(* Init ST03_513_B70_2 Führungsschiene  Zuführung Stopper AST (ValveSensor) *)
ST03_513_B70_2.sInit.InstName		:='ST03_513_B70_2';
ST03_513_B70_2.sInit.BitName		:='+8_512_B70.2';
ST03_513_B70_2.sInit.Description	:='Führungsschiene  Zuführung Stopper AST';
ST03_513_B70_2.sInit.SensorType	:=sValveSensorType_WORK;

(* Init ST03_513_B70_3 Führungsschiene  Zuführung Stopper GST (ValveSensor) *)
ST03_513_B70_3.sInit.InstName		:='ST03_513_B70_3';
ST03_513_B70_3.sInit.BitName		:='+8_513_B70.3';
ST03_513_B70_3.sInit.Description	:='Führungsschiene  Zuführung Stopper GST';
ST03_513_B70_3.sInit.SensorType	:=sValveSensorType_INIT;

(* Init ST03_513_B70_4 ISK anwesend am Stoper (DigIn) *)
ST03_513_B70_4.sInit.InstName            :='ST03_513_B70_4';
ST03_513_B70_4.sInit.Description         :='ISK anwesend am Stoper';
ST03_513_B70_4.sInit.BitInName           :='+8-513_B670.4';
ST03_513_B70_4.sInit.HomePosSignal       :=2; (* 0: Signal=Low, 1: Signal=High, 2: always  *)
ST03_513_B70_4.sInit.MaxTime             :=2000;
ST03_513_B70_4.sInit.EnableInEveryMode   :=TRUE;

(* Init ST03_513_B70_5 Übergabeposition Stopper 1 AST (ValveSensor) *)
ST03_513_B70_5.sInit.InstName		:='ST03_513_B70_5';
ST03_513_B70_5.sInit.BitName		:='+8_513_B70.5';
ST03_513_B70_5.sInit.Description	:='Übergabeposition Stopper 1 AST';
ST03_513_B70_5.sInit.SensorType	:=sValveSensorType_WORK;

(* Init ST03_513_B70_6 Übergabeposition Stopper 1 GST (ValveSensor) *)
ST03_513_B70_6.sInit.InstName		:='ST03_513_B70_6';
ST03_513_B70_6.sInit.BitName		:='+8_513_B70.6';
ST03_513_B70_6.sInit.Description	:='Übergabeposition Stopper 1 GST';
ST03_513_B70_6.sInit.SensorType	:=sValveSensorType_INIT;

(* Init ST03_513_B70_7 ISK auf Übergabeposition 1 (DigIn) *)
ST03_513_B70_7.sInit.InstName            :='ST03_513_B70_7';
ST03_513_B70_7.sInit.Description         :='ISK auf Übergabeposition 1';
ST03_513_B70_7.sInit.BitInName           :='+8-513_B670.7';
ST03_513_B70_7.sInit.HomePosSignal       :=2; (* 0: Signal=Low, 1: Signal=High, 2: always  *)
ST03_513_B70_7.sInit.MaxTime             :=2000;
ST03_513_B70_7.sInit.EnableInEveryMode   :=TRUE;


(* Init ST03_514_B71_0 Übergabeposition Stopper 2 AST (ValveSensor) *)
ST03_514_B71_0.sInit.InstName		:='ST03_514_B71_0';
ST03_514_B71_0.sInit.BitName		:='+8_514_B71.0';
ST03_514_B71_0.sInit.Description	:='Übergabeposition Stopper 2 AST';
ST03_514_B71_0.sInit.SensorType	:=sValveSensorType_WORK;

(* Init ST03_514_B71_1 Übergabeposition Stopper 2 GST (ValveSensor) *)
ST03_514_B71_1.sInit.InstName		:='ST03_514_B71_1';
ST03_514_B71_1.sInit.BitName		:='+8_514_B71.1';
ST03_514_B71_1.sInit.Description	:='Übergabeposition Stopper 2 GST';
ST03_514_B71_1.sInit.SensorType	:=sValveSensorType_INIT;

(* Init ST03_514_B71_2 ISK auf Übergabeposition 2 (DigIn) *)
ST03_514_B71_2.sInit.InstName            :='ST03_514_B71_2';
ST03_514_B71_2.sInit.Description         :='ISK auf Übergabeposition 2';
ST03_514_B71_2.sInit.BitInName           :='+8-514_B71.2';
ST03_514_B71_2.sInit.HomePosSignal       :=2; (* 0: Signal=Low, 1: Signal=High, 2: always  *)
ST03_514_B71_2.sInit.MaxTime             :=2000;
ST03_514_B71_2.sInit.EnableInEveryMode   :=TRUE;

(* Init ST03_514_B71_3 Übergabeposition Stopper 3 AST (ValveSensor) *)
ST03_514_B71_3.sInit.InstName		:='ST03_514_B71_3';
ST03_514_B71_3.sInit.BitName		:='+8_514_B71.3';
ST03_514_B71_3.sInit.Description	:='Übergabeposition Stopper 3 AST';
ST03_514_B71_3.sInit.SensorType	:=sValveSensorType_WORK;

(* Init ST03_514_B71_4 Übergabeposition Stopper 3 GST (ValveSensor) *)
ST03_514_B71_4.sInit.InstName		:='ST03_514_B71_4';
ST03_514_B71_4.sInit.BitName		:='+8_514_B71.4';
ST03_514_B71_4.sInit.Description	:='Übergabeposition Stopper 3 GST';
ST03_514_B71_4.sInit.SensorType	:=sValveSensorType_INIT;

(* Init ST03_514_B71_5 ISK auf Übergabeposition 3 (DigIn) *)
ST03_514_B71_5.sInit.InstName            :='ST03_514_B71_5';
ST03_514_B71_5.sInit.Description         :='ISK auf Übergabeposition 3';
ST03_514_B71_5.sInit.BitInName           :='+8-514_B71.5';
ST03_514_B71_5.sInit.HomePosSignal       :=2; (* 0: Signal=Low, 1: Signal=High, 2: always  *)
ST03_514_B71_5.sInit.MaxTime             :=2000;
ST03_514_B71_5.sInit.EnableInEveryMode   :=TRUE;

(* Init ST03_514_B71_6 ISK auf Übergabeposition 4 (DigIn) *)
ST03_514_B71_6.sInit.InstName            :='ST03_514_B71_6';
ST03_514_B71_6.sInit.Description         :='ISK auf Übergabeposition 4';
ST03_514_B71_6.sInit.BitInName           :='+8-514_B71.6';
ST03_514_B71_6.sInit.HomePosSignal       :=2; (* 0: Signal=Low, 1: Signal=High, 2: always  *)
ST03_514_B71_6.sInit.MaxTime             :=2000;
ST03_514_B71_6.sInit.EnableInEveryMode   :=TRUE;

(* Init ST03_514_B71_7 Führungsschiene frei zum schwenken (DigIn) *)
ST03_514_B71_7.sInit.InstName            :='ST03_514_B71_7';
ST03_514_B71_7.sInit.Description         :='Führungsschiene frei zum schwenken';
ST03_514_B71_7.sInit.BitInName           :='+8-514_B71.7';
ST03_514_B71_7.sInit.HomePosSignal       :=2; (* 0: Signal=Low, 1: Signal=High, 2: always  *)
ST03_514_B71_7.sInit.MaxTime             :=2000;
ST03_514_B71_7.sInit.EnableInEveryMode   :=TRUE;

(* Init ST03_515_Y72_0   ISK Klemmer 1 AST/GST (Valve) *)
ST03_515_Y72_0.sInit.InstName            :='ST03_515_Y72_0';
ST03_515_Y72_0.sInit.BitName            :='+8-515_Y72.0';
ST03_515_Y72_0.sInit.Description         :=' ISK Klemmer 1 AST/GST';
ST03_515_Y72_0.sInit.HomePosDefine       :=HOME_ALWAYS;
ST03_515_Y72_0.sInit.InitDescription     :='GS auf';
ST03_515_Y72_0.sInit.WorkDescription     :='AS zu';
(*ST03_515_Y72_0.sInit.InitDescription     :='GS zu';
ST03_515_Y72_0.sInit.WorkDescription     :='AS auf';*)
ST03_515_Y72_0.sInit.DampBothTime        :=200;
ST03_515_Y72_0.sInit.KindOfValve         :='A';
ST03_515_Y72_0.sInit.MaxTime             :=2000;

(* Init ST03_515_Y72_1  Rinne schwenkern  AST/GST (Valve) *)
ST03_515_Y72_1.sInit.InstName            :='ST03_515_Y72_1';
ST03_515_Y72_1.sInit.BitName            :='+8-515_Y72.1';
ST03_515_Y72_1.sInit.Description         :=' Rinne schwenkern AST/GST';
ST03_515_Y72_1.sInit.HomePosDefine       :=HOME_ALWAYS;
ST03_515_Y72_1.sInit.InitDescription     :='GS 0 Grad';
ST03_515_Y72_1.sInit.WorkDescription     :='AS 180 Grad';
ST03_515_Y72_1.sInit.DampBothTime        :=200;
ST03_515_Y72_1.sInit.KindOfValve         :='A';
ST03_515_Y72_1.sInit.MaxTime             :=2000;

(* Init ST03_515_Y72_2  Führungsschiene  Zuführung Vereinzler   AST/GST (Valve) *)
ST03_515_Y72_2.sInit.InstName            :='ST03_515_Y72_2';
ST03_515_Y72_2.sInit.BitName            :='+8-515_Y72.2';
ST03_515_Y72_2.sInit.Description         :=' Führungsschiene  Zuführung Vereinzler AST/GST';
ST03_515_Y72_2.sInit.HomePosDefine       :=HOME_ALWAYS;
ST03_515_Y72_2.sInit.InitDescription     :='GS auf';
ST03_515_Y72_2.sInit.WorkDescription     :='AS zu';
ST03_515_Y72_2.sInit.DampBothTime        :=200;
ST03_515_Y72_2.sInit.KindOfValve         :='A';
ST03_515_Y72_2.sInit.MaxTime             :=2000;

(* Init ST03_515_Y72_3  Führungsschiene  Zuführung Stopper   AST/GST (Valve) *)
ST03_515_Y72_3.sInit.InstName            :='ST03_515_Y72_3';
ST03_515_Y72_3.sInit.BitName            :='+8-515_Y72.3';
ST03_515_Y72_3.sInit.Description         :=' Führungsschiene  Zuführung Stopper AST/GST';
ST03_515_Y72_3.sInit.HomePosDefine       :=HOME_ALWAYS;
ST03_515_Y72_3.sInit.InitDescription     :='GS ausfahren';
ST03_515_Y72_3.sInit.WorkDescription     :='AS einfahren';
ST03_515_Y72_3.sInit.DampBothTime        :=200;
ST03_515_Y72_3.sInit.KindOfValve         :='A';
ST03_515_Y72_3.sInit.MaxTime             :=2000;

(* Init ST03_515_Y72_4  Übergabeposition Stopper 1   AST/GST (Valve) *)
ST03_515_Y72_4.sInit.InstName            :='ST03_515_Y72_4';
ST03_515_Y72_4.sInit.BitName            :='+8-515_Y72.4';
ST03_515_Y72_4.sInit.Description         :=' Übergabeposition Stopper 1 AST/GST';
ST03_515_Y72_4.sInit.HomePosDefine       :=HOME_ALWAYS;
ST03_515_Y72_4.sInit.InitDescription     :='GS ausfahren';
ST03_515_Y72_4.sInit.WorkDescription     :='AS einfahren';
ST03_515_Y72_4.sInit.DampBothTime        :=200;
ST03_515_Y72_4.sInit.KindOfValve         :='A';
ST03_515_Y72_4.sInit.MaxTime             :=2000;

(* Init ST03_515_Y72_5  Übergabeposition Stopper 2   AST/GST (Valve) *)
ST03_515_Y72_5.sInit.InstName            :='ST03_515_Y72_5';
ST03_515_Y72_5.sInit.BitName            :='+8-515_Y72.5';
ST03_515_Y72_5.sInit.Description         :=' Übergabeposition Stopper 2 AST/GST';
ST03_515_Y72_5.sInit.HomePosDefine       :=HOME_ALWAYS;
ST03_515_Y72_5.sInit.InitDescription     :='GS ausfahren';
ST03_515_Y72_5.sInit.WorkDescription     :='AS einfahren';
ST03_515_Y72_5.sInit.DampBothTime        :=200;
ST03_515_Y72_5.sInit.KindOfValve         :='A';
ST03_515_Y72_5.sInit.MaxTime             :=2000;

(* Init ST03_515_Y72_6  Übergabeposition Stopper 3   AST/GST (Valve) *)
ST03_515_Y72_6.sInit.InstName            :='ST03_515_Y72_6';
ST03_515_Y72_6.sInit.BitName            :='+8-515_Y72.6';
ST03_515_Y72_6.sInit.Description         :=' Übergabeposition Stopper 3 AST/GST';
ST03_515_Y72_6.sInit.HomePosDefine       :=HOME_ALWAYS;
ST03_515_Y72_6.sInit.InitDescription     :='GS ausfahren';
ST03_515_Y72_6.sInit.WorkDescription     :='AS einfahren';
ST03_515_Y72_6.sInit.DampBothTime        :=200;
ST03_515_Y72_6.sInit.KindOfValve         :='A';
ST03_515_Y72_6.sInit.MaxTime             :=2000;
END_ACTION
ACTION Init_88pol:
(*Rüstsatz 88 pol==================================================================================*)

(* Init ST03_501_B69_0 Zuführung  frei zum Ablegen ISK SP Maschine (DigIn) *)
ST03_501_B69_0.sInit.InstName            :='ST03_501_B69_0';
ST03_501_B69_0.sInit.Description         :='frei zum Ablegen ISK SP Maschine';
ST03_501_B69_0.sInit.BitInName           :='+8-501_B69.0';
ST03_501_B69_0.sInit.HomePosSignal       :=2; (* 0: Signal=Low, 1: Signal=High, 2: always  *)
ST03_501_B69_0.sInit.MaxTime             :=2000;
ST03_501_B69_0.sInit.EnableInEveryMode   :=TRUE;

(* Init ST03_501_B69_1 Zuführung Vereinzler AST (ValveSensor) *)
ST03_501_B69_1.sInit.InstName		:='ST03_501_B69_1';
ST03_501_B69_1.sInit.BitName		:='+8_501_B69.1';
ST03_501_B69_1.sInit.Description	:='Zuführung Vereinzler AST';
ST03_501_B69_1.sInit.SensorType	:=sValveSensorType_WORK;

(* Init ST03_501_B69_2 Zuführung Vereinzler GST (ValveSensor) *)
ST03_501_B69_2.sInit.InstName		:='ST03_501_B69_2';
ST03_501_B69_2.sInit.BitName		:='+8_501_B69.2';
ST03_501_B69_2.sInit.Description	:='Zuführung Vereinzler GST';
ST03_501_B69_2.sInit.SensorType	:=sValveSensorType_INIT;

(* Init ST03_501_B69_3 Zuführung Stopper AST (ValveSensor) *)
ST03_501_B69_3.sInit.InstName		:='ST03_501_B69_3';
ST03_501_B69_3.sInit.BitName		:='+8_501_B69.3';
ST03_501_B69_3.sInit.Description	:='Zuführung Stopper AST';
ST03_501_B69_3.sInit.SensorType	:=sValveSensorType_WORK;

(* Init ST03_501_B69_4 Zuführung Stopper GST (ValveSensor) *)
ST03_501_B69_4.sInit.InstName		:='ST03_501_B69_4';
ST03_501_B69_4.sInit.BitName		:='+8_501_B69.4';
ST03_501_B69_4.sInit.Description	:='Zuführung Stopper GST';
ST03_501_B69_4.sInit.SensorType	:=sValveSensorType_INIT;

(* Init ST03_501_B69_5 ISK anwesend am Vereinzler (DigIn) *)
ST03_501_B69_5.sInit.InstName            :='ST03_501_B69_5';
ST03_501_B69_5.sInit.Description         :='ISK anwesend am Vereinzler';
ST03_501_B69_5.sInit.BitInName           :='+8-501_B69.5';
ST03_501_B69_5.sInit.HomePosSignal       :=2; (* 0: Signal=Low, 1: Signal=High, 2: always  *)
ST03_501_B69_5.sInit.MaxTime             :=2000;
ST03_501_B69_5.sInit.EnableInEveryMode   :=TRUE;

(* Init ST03_501_B69_6 ISK anwesend am Stopper (DigIn) *)
ST03_501_B69_6.sInit.InstName            :='ST03_501_B69_6';
ST03_501_B69_6.sInit.Description         :='ISK anwesend am Stopper';
ST03_501_B69_6.sInit.BitInName           :='+8-501_B69.6';
ST03_501_B69_6.sInit.HomePosSignal       :=2; (* 0: Signal=Low, 1: Signal=High, 2: always  *)
ST03_501_B69_6.sInit.MaxTime             :=2000;
ST03_501_B69_6.sInit.EnableInEveryMode   :=TRUE;

(* Init ST03_501_B69_7 ISK auf Abholposition Robi (DigIn) *)
ST03_501_B69_7.sInit.InstName            :='ST03_501_B69_7';
ST03_501_B69_7.sInit.Description         :='ISK auf Abholposition Robi';
ST03_501_B69_7.sInit.BitInName           :='+8-501_B69.7';
ST03_501_B69_7.sInit.HomePosSignal       :=2; (* 0: Signal=Low, 1: Signal=High, 2: always  *)
ST03_501_B69_7.sInit.MaxTime             :=2000;
ST03_501_B69_7.sInit.EnableInEveryMode   :=TRUE;

(* Init ST03_502_B70_0 ISK Lageerkennung(DigIn) *)
ST03_502_B70_0.sInit.InstName            :='ST03_502_B70_0';
ST03_502_B70_0.sInit.Description         :='ISK Lageerkennung';
ST03_502_B70_0.sInit.BitInName           :='+8-502_B70.0';
ST03_502_B70_0.sInit.HomePosSignal       :=2; (* 0: Signal=Low, 1: Signal=High, 2: always  *)
ST03_502_B70_0.sInit.MaxTime             :=2000;
ST03_502_B70_0.sInit.EnableInEveryMode   :=TRUE;

(* Init ST03_502_Y70_1  Zuführung  Vereinzler AST/GST (Valve) *)
ST03_502_Y70_1.sInit.InstName            :='ST03_502_Y70_1';
ST03_502_Y70_1.sInit.BitName            :='+8-502_Y70.1';
ST03_502_Y70_1.sInit.Description         :=' Zuführung Vereinzler AST/GST';
ST03_502_Y70_1.sInit.HomePosDefine       :=HOME_ALWAYS;
ST03_502_Y70_1.sInit.InitDescription     :='GS einfahren';
ST03_502_Y70_1.sInit.WorkDescription     :='AS ausfahren';
ST03_502_Y70_1.sInit.DampBothTime        :=200;
ST03_502_Y70_1.sInit.KindOfValve         :='A';
ST03_502_Y70_1.sInit.MaxTime             :=2000;

(* Init ST03_502_Y70_2  Zuführung  Stopper AST/GST (Valve) *)
ST03_502_Y70_2.sInit.InstName            :='ST03_502_Y70_2';
ST03_502_Y70_2.sInit.BitName            :='+8-502_Y70.2';
ST03_502_Y70_2.sInit.Description         :=' Zuführung Stopper AST/GST';
ST03_502_Y70_2.sInit.HomePosDefine       :=HOME_ALWAYS;
ST03_502_Y70_2.sInit.InitDescription     :='GS ausfahren';
ST03_502_Y70_2.sInit.WorkDescription     :='AS einfahren';
ST03_502_Y70_2.sInit.DampBothTime        :=200;
ST03_502_Y70_2.sInit.KindOfValve         :='A';
ST03_502_Y70_2.sInit.MaxTime             :=2000;
END_ACTION
ACTION Init_88polAMG:
(*Rüstsatz 88 pol AMG==================================================================================*)

(* Init ST03_521_B69_0 Zuführung  frei zum Ablegen ISK SP Maschine (DigIn) *)
ST03_521_B69_0.sInit.InstName            :='ST03_521_B69_0';
ST03_521_B69_0.sInit.Description         :='frei zum Ablegen ISK SP Maschine';
ST03_521_B69_0.sInit.BitInName           :='+8-521_B69.0';
ST03_521_B69_0.sInit.HomePosSignal	:=2; (* 0: Signal=Low, 1: Signal=High, 2: always  *)
ST03_521_B69_0.sInit.MaxTime             :=2000;
ST03_521_B69_0.sInit.EnableInEveryMode   :=TRUE;

(* Init ST03_521_B69_1 Zuführung Vereinzler eingefahren GST (ValveSensor) *)
ST03_521_B69_1.sInit.InstName		:='ST03_521_B69_1';
ST03_521_B69_1.sInit.BitName		:='+8_521_B69.1';
ST03_521_B69_1.sInit.Description	:=' Vereinzler eingefahren GST';
ST03_521_B69_1.sInit.SensorType	:=sValveSensorType_INIT;

(* Init ST03_521_B69_2 Zuführung Vereinzler ausgefahren AST (ValveSensor) *)
ST03_521_B69_2.sInit.InstName		:='ST03_521_B69_2';
ST03_521_B69_2.sInit.BitName		:='+8_521_B69.2';
ST03_521_B69_2.sInit.Description	:=' Vereinzler ausgefahren AST';
ST03_521_B69_2.sInit.SensorType	:=sValveSensorType_WORK;

(* Init ST03_521_B69_3 Zuführung Stopper eingefahren AST (ValveSensor) *)
ST03_521_B69_3.sInit.InstName		:='ST03_521_B69_3';
ST03_521_B69_3.sInit.BitName		:='+8_521_B69.3';
ST03_521_B69_3.sInit.Description	:='Stopper eingefahren AST';
ST03_521_B69_3.sInit.SensorType	:=sValveSensorType_WORK;

(* Init ST03_521_B69_4 Zuführung Stopper ausgefahren GST (ValveSensor) *)
ST03_521_B69_4.sInit.InstName		:='ST03_521_B69_4';
ST03_521_B69_4.sInit.BitName		:='+8_521_B69.4';
ST03_521_B69_4.sInit.Description	:='Stopper ausgefahren GST';
ST03_521_B69_4.sInit.SensorType	:=sValveSensorType_INIT;;

(* Init ST03_521_B69_6 ISK anwesend am Stopper (DigIn) *)
ST03_521_B69_6.sInit.InstName            :='ST03_521_B69_6';
ST03_521_B69_6.sInit.Description         :='ISK anwesend am Stopper';
ST03_521_B69_6.sInit.BitInName           :='+8-521_B69.6';
ST03_521_B69_6.sInit.HomePosSignal       :=2; (* 0: Signal=Low, 1: Signal=High, 2: always  *)
ST03_521_B69_6.sInit.MaxTime             :=2000;
ST03_521_B69_6.sInit.EnableInEveryMode   :=TRUE;

(* Init ST03_521_B69_7 ISK Lageerkennung links (DigIn) *)
ST03_521_B69_7.sInit.InstName            :='ST03_521_B69_7';
ST03_521_B69_7.sInit.Description         :='ISK Lageerkennung links';
ST03_521_B69_7.sInit.BitInName           :='+8-521_B69.7';
ST03_521_B69_7.sInit.HomePosSignal       :=2; (* 0: Signal=Low, 1: Signal=High, 2: always  *)
ST03_521_B69_7.sInit.MaxTime             :=2000;
ST03_521_B69_7.sInit.EnableInEveryMode   :=TRUE;

(* Init ST03_522_B70_0 SK Lageerkennung rechts(DigIn) *)
ST03_522_B70_0.sInit.InstName            :='ST03_522_B70_0';
ST03_522_B70_0.sInit.Description         :='ISK Lageerkennung rechts';
ST03_522_B70_0.sInit.BitInName           :='+8-522_B70.0';
ST03_522_B70_0.sInit.HomePosSignal       :=2; (* 0: Signal=Low, 1: Signal=High, 2: always  *)
ST03_522_B70_0.sInit.MaxTime             :=2000;
ST03_522_B70_0.sInit.EnableInEveryMode   :=TRUE;

(* Init ST03_522_Y70_1   Zuführung  Vereinzler AST/GST (Valve) *)
ST03_522_Y70_1.sInit.InstName            :='ST03_522_Y70_1';
ST03_522_Y70_1.sInit.BitName            :='+8-522_Y70.1';
ST03_522_Y70_1.sInit.Description         :=' Zuführung Vereinzler AST/GST';
ST03_522_Y70_1.sInit.HomePosDefine       :=HOME_ALWAYS;
ST03_522_Y70_1.sInit.InitDescription     :='GS einfahren';
ST03_522_Y70_1.sInit.WorkDescription     :='AS ausfahren';
ST03_522_Y70_1.sInit.DampBothTime        :=200;
ST03_522_Y70_1.sInit.KindOfValve         :='A';
ST03_522_Y70_1.sInit.MaxTime             :=2000;

(* Init ST03_522_Y70_2   Zuführung  Stopper AST/GST (Valve) *)
ST03_522_Y70_2.sInit.InstName            :='ST03_522_Y70_2';
ST03_522_Y70_2.sInit.BitName            :='+8-522_Y70.2';
ST03_522_Y70_2.sInit.Description         :=' Zuführung Stopper AST/GST';
ST03_522_Y70_2.sInit.HomePosDefine       :=HOME_ALWAYS;
ST03_522_Y70_2.sInit.InitDescription     :='GS ausfahren';
ST03_522_Y70_2.sInit.WorkDescription     :='AS einfahren';
ST03_522_Y70_2.sInit.DampBothTime        :=200;
ST03_522_Y70_2.sInit.KindOfValve         :='A';
ST03_522_Y70_2.sInit.MaxTime             :=2000;
END_ACTION
ACTION Init_92pol:
(*Rüstsatz 92pol*)
(* Init ST03_444_B69_0 Förderbandeinheit  Zuführung Vereinzler AST (ValveSensor) *)
ST03_444_B69_0.sInit.InstName            :='ST03_444_B69_0';
ST03_444_B69_0.sInit.BitName            :='+8_444_B69.0';
ST03_444_B69_0.sInit.Description         :='Förderbandeinheit  Zuführung Vereinzler AST';
ST03_444_B69_0.sInit.SensorType          :=sValveSensorType_INIT;

(* Init ST03_444_B69_1 Förderbandeinheit  Zuführung Vereinzler GST (ValveSensor) *)
ST03_444_B69_1.sInit.InstName            :='ST03_444_B69_1';
ST03_444_B69_1.sInit.BitName            :='+8_444_B69.1';
ST03_444_B69_1.sInit.Description         :='Förderbandeinheit  Zuführung Vereinzler GST';
ST03_444_B69_1.sInit.SensorType          :=sValveSensorType_WORK;

(* Init ST03_444_B69_2 Förderbandeinheit  Zuführung Stopper AST (ValveSensor) *)
ST03_444_B69_2.sInit.InstName            :='ST03_444_B69_2';
ST03_444_B69_2.sInit.BitName            :='+8_444_B69.2';
ST03_444_B69_2.sInit.Description         :='Förderband linke Zuführung Stopper AST';
ST03_444_B69_2.sInit.SensorType          :=sValveSensorType_INIT;

(* Init ST03_444_B69_3 Förderbandeinheit  Zuführung Stopper GST (ValveSensor) *)
ST03_444_B69_3.sInit.InstName            :='ST03_444_B69_3';
ST03_444_B69_3.sInit.BitName            :='+8_444_B69.3';
ST03_444_B69_3.sInit.Description         :='Förderband linke Zuführung Stopper GST';
ST03_444_B69_3.sInit.SensorType          :=sValveSensorType_WORK;

(* Init ST03_444_B69_4  Zuführung  frei zum Ablegen ISK SP Maschine Pos.1 (DigIn) *)
ST03_444_B69_4.sInit.InstName            :='ST03_444_B69_4';
ST03_444_B69_4.sInit.Description         :='Zuführung links frei zum Ablegen ISK SP Maschine Pos1';
ST03_444_B69_4.sInit.BitInName           :='+8-444_B69.4';
ST03_444_B69_4.sInit.HomePosSignal       :=2; (* 0: Signal=Low, 1: Signal=High, 2: always  *)
ST03_444_B69_4.sInit.MaxTime             :=2000;
ST03_444_B69_4.sInit.EnableInEveryMode   :=TRUE;

(* Init ST03_444_B69_7  ISK anwesend am Vereinzler (DigIn) *)
ST03_444_B69_7.sInit.InstName            :='ST03_444_B69_7';
ST03_444_B69_7.sInit.Description         :='ISK anwesend am Vereinzler';
ST03_444_B69_7.sInit.BitInName           :='+8-444_B69.7';
ST03_444_B69_7.sInit.HomePosSignal       :=2; (* 0: Signal=Low, 1: Signal=High, 2: always  *)
ST03_444_B69_7.sInit.MaxTime             :=2000;
ST03_444_B69_7.sInit.EnableInEveryMode   :=TRUE;

(* Init ST03_445_B70_1  Züführung  ISK Lageerkennung 1 (DigIn) *)
ST03_445_B70_1.sInit.InstName            :='ST03_445_B70_1';
ST03_445_B70_1.sInit.Description         :='Züführung  ISK Lageerkennung 1';
ST03_445_B70_1.sInit.BitInName           :='+8-445_B70.1';
ST03_445_B70_1.sInit.HomePosSignal       :=2; (* 0: Signal=Low, 1: Signal=High, 2: always  *)
ST03_445_B70_1.sInit.MaxTime             :=2000;
ST03_445_B70_1.sInit.EnableInEveryMode   :=TRUE;

(* Init ST03_445_B70_2  Züführung  ISK Lageerkennung 2 (DigIn) *)
ST03_445_B70_2.sInit.InstName            :='ST03_445_B70_2';
ST03_445_B70_2.sInit.Description         :='Züführung  ISK Lageerkennung 2';
ST03_445_B70_2.sInit.BitInName           :='+8-445_B70.2';
ST03_445_B70_2.sInit.HomePosSignal       :=2; (* 0: Signal=Low, 1: Signal=High, 2: always  *)
ST03_445_B70_2.sInit.MaxTime             :=2000;
ST03_445_B70_2.sInit.EnableInEveryMode   :=TRUE;

(* Init ST03_446_B70_4  ISK anwesend Übergabeposition Roboter (DigIn) *)
ST03_446_B70_4.sInit.InstName            :='ST03_446_B70_4';
ST03_446_B70_4.sInit.Description         :='Zuführung ISK auf Übergabeposition Robo Palettierer ';
ST03_446_B70_4.sInit.BitInName           :='+8-446_B70.4';
ST03_446_B70_4.sInit.HomePosSignal       :=2; (* 0: Signal=Low, 1: Signal=High, 2: always  *)
ST03_446_B70_4.sInit.MaxTime             :=2000;
ST03_446_B70_4.sInit.EnableInEveryMode   :=TRUE;

(* Init ST03_446_Y70_5 Förderband  Zuführung Vereinzler (Valve) *)
ST03_446_Y70_5.sInit.InstName            :='ST03_446_Y70_5';
ST03_446_Y70_5.sInit.BitName            :='+8-446_Y70.5';
ST03_446_Y70_5.sInit.Description         :='Förderband  Zuführung Vereinzler';
ST03_446_Y70_5.sInit.HomePosDefine       :=HOME_ALWAYS;
ST03_446_Y70_5.sInit.InitDescription     :='GS einfahren';
ST03_446_Y70_5.sInit.WorkDescription     :='AS ausfahren';
ST03_446_Y70_5.sInit.DampBothTime        :=200;
ST03_446_Y70_5.sInit.KindOfValve         :='A';
ST03_446_Y70_5.sInit.MaxTime             :=2000;

(* Init ST03_446_Y70_6 Förderband  Zuführung Stopper (Valve) *)
ST03_446_Y70_6.sInit.InstName            :='ST03_446_Y70_6';
ST03_446_Y70_6.sInit.BitName            :='+8-446_Y70.6';
ST03_446_Y70_6.sInit.Description         :='Förderband  Zuführung Stopper';
ST03_446_Y70_6.sInit.HomePosDefine       :=HOME_ALWAYS;
ST03_446_Y70_6.sInit.InitDescription     :='GS ausfahren';
ST03_446_Y70_6.sInit.WorkDescription     :='AS einfahren';
ST03_446_Y70_6.sInit.DampBothTime        :=200;
ST03_446_Y70_6.sInit.KindOfValve         :='A';
ST03_446_Y70_6.sInit.MaxTime             :=2000;
END_ACTION
ACTION Init_NOX4pol:
(*Rüstsatz NOX 4 pol==================================================================================*)

(* Init ST03_491_B69_0 Zuführung  frei zum Ablegen ISK SP Maschine (DigIn) *)
ST03_491_B69_0.sInit.InstName            :='ST03_491_B69_0';
ST03_491_B69_0.sInit.Description         :='frei zum Ablegen ISK SP Maschine';
ST03_491_B69_0.sInit.BitInName           :='+8-491_B69.0';
ST03_491_B69_0.sInit.HomePosSignal       :=2; (* 0: Signal=Low, 1: Signal=High, 2: always  *)
ST03_491_B69_0.sInit.MaxTime             :=2000;
ST03_491_B69_0.sInit.EnableInEveryMode   :=TRUE;

(* Init ST03_491_B69_5 ISK anwesend am Stoper (DigIn) *)
ST03_491_B69_5.sInit.InstName            :='ST03_491_B69_5';
ST03_491_B69_5.sInit.Description         :='ISK anwesend am Stoper';
ST03_491_B69_5.sInit.BitInName           :='+8-491_B69.5';
ST03_491_B69_5.sInit.HomePosSignal       :=2; (* 0: Signal=Low, 1: Signal=High, 2: always  *)
ST03_491_B69_5.sInit.MaxTime             :=2000;
ST03_491_B69_5.sInit.EnableInEveryMode   :=TRUE;

(* Init ST03_491_B69_7 SK auf Abholposition Robi (DigIn) *)
ST03_491_B69_7.sInit.InstName            :='ST03_491_B69_7';
ST03_491_B69_7.sInit.Description         :='SK auf Abholposition Robi';
ST03_491_B69_7.sInit.BitInName           :='+8-491_B69.5';
ST03_491_B69_7.sInit.HomePosSignal       :=2; (* 0: Signal=Low, 1: Signal=High, 2: always  *)
ST03_491_B69_7.sInit.MaxTime             :=2000;
ST03_491_B69_7.sInit.EnableInEveryMode   :=TRUE;

(* Init ST03_492_Y70_0  Zuführung Vereinzler AST/GST (Valve) *)
ST03_492_Y70_0.sInit.InstName            :='ST03_492_Y70_0';
ST03_492_Y70_0.sInit.BitName            :='+8-492_Y70.0';
ST03_492_Y70_0.sInit.Description         :='Zuführung Vereinzler AST/GST';
ST03_492_Y70_0.sInit.HomePosDefine       :=HOME_ALWAYS;
ST03_492_Y70_0.sInit.InitDescription     :='GS einfahren';
ST03_492_Y70_0.sInit.WorkDescription     :='AS ausfahren';
ST03_492_Y70_0.sInit.DampBothTime        :=200;
ST03_492_Y70_0.sInit.KindOfValve         :='A';
ST03_492_Y70_0.sInit.MaxTime             :=2000;

(* Init ST03_491_B69_1 Zuführung Vereinzler AST (ValveSensor) *)
ST03_491_B69_1.sInit.InstName		:='ST03_491_B69_1';
ST03_491_B69_1.sInit.BitName		:='+8_491_B69.1';
ST03_491_B69_1.sInit.Description	:='Zuführung  Vereinzler AST';
ST03_491_B69_1.sInit.SensorType	:=sValveSensorType_WORK;

(* Init ST03_491_B69_2 Zuführung Vereinzler GST (ValveSensor) *)
ST03_491_B69_2.sInit.InstName		:='ST03_491_B69_2';
ST03_491_B69_2.sInit.BitName		:='+8_491_B69.2';
ST03_491_B69_2.sInit.Description	:='Zuführung Vereinzler GST';
ST03_491_B69_2.sInit.SensorType	:=sValveSensorType_INIT;

(* Init ST03_492_Y70_1   Zuführung  Stopper AST/GST (Valve) *)
ST03_492_Y70_1.sInit.InstName            :='ST03_492_Y70_1';
ST03_492_Y70_1.sInit.BitName            :='+8-492_Y70.1';
ST03_492_Y70_1.sInit.Description         :=' Zuführung Stopper AST/GST';
ST03_492_Y70_1.sInit.HomePosDefine       :=HOME_ALWAYS;
ST03_492_Y70_1.sInit.InitDescription     :='GS ausfahren';
ST03_492_Y70_1.sInit.WorkDescription     :='AS einfahren';
ST03_492_Y70_1.sInit.DampBothTime        :=200;
ST03_492_Y70_1.sInit.KindOfValve         :='A';
ST03_492_Y70_1.sInit.MaxTime             :=2000;

(* Init ST03_491_B69_3 Zuführung Stopper AST (ValveSensor) *)
ST03_491_B69_3.sInit.InstName		:='ST03_491_B69_3';
ST03_491_B69_3.sInit.BitName		:='+8_491_B69.3';
ST03_491_B69_3.sInit.Description	:='Zuführung Stopper AST';
ST03_491_B69_3.sInit.SensorType	:=sValveSensorType_WORK;

(* Init ST03_491_B69_4 Zuführung Stopper GST (ValveSensor) *)
ST03_491_B69_4.sInit.InstName		:='ST03_491_B69_4';
ST03_491_B69_4.sInit.BitName		:='+8_491_B69.4';
ST03_491_B69_4.sInit.Description	:='Zuführung Stopper GST';
ST03_491_B69_4.sInit.SensorType	:=sValveSensorType_INIT;
END_ACTION
ACTION Init_NOX5_6pol:
(*===============================Rüstsatz NOX 5+6 pol==========================*)

(* Init ST03_4x2_B69_0 Zuführung frei zum Ablegen ISK SP Maschine (DigIn) *)
ST03_4x2_B69_0.sInit.InstName            :='ST03_4x2_B69_0';
ST03_4x2_B69_0.sInit.Description         :='Zuführung frei zum Ablegen ISK SP Maschine';
ST03_4x2_B69_0.sInit.BitInName           :='+8-4x2_B69.0';
ST03_4x2_B69_0.sInit.HomePosSignal       :=2; (* 0: Signal=Low, 1: Signal=High, 2: always  *)
ST03_4x2_B69_0.sInit.MaxTime             :=2000;
ST03_4x2_B69_0.sInit.EnableInEveryMode   :=TRUE;

(* Init ST03_4x2_B69_1 Zuführung Vereinzler GST eingefahren (ValveSensor) *)
ST03_4x2_B69_1.sInit.InstName		:='ST03_4x2_B69_1';
ST03_4x2_B69_1.sInit.BitName		:='+8_4x2_B69.1';
ST03_4x2_B69_1.sInit.Description	:='Zuführung Vereinzler GST';
ST03_4x2_B69_1.sInit.SensorType		:=sValveSensorType_INIT;

(* Init ST03_4x2_B69_2 Zuführung Vereinzler AST ausgefahren (ValveSensor) *)
ST03_4x2_B69_2.sInit.InstName		:='ST03_4x2_B69_2';
ST03_4x2_B69_2.sInit.BitName		:='+8_4x2_B69.2';
ST03_4x2_B69_2.sInit.Description	:='Zuführung Vereinzler AST';
ST03_4x2_B69_2.sInit.SensorType		:=sValveSensorType_WORK;

(* Init ST03_4x2_B69_3 Zuführung Stopper GST eingefahren (ValveSensor) *)
ST03_4x2_B69_3.sInit.InstName		:='ST03_4x2_B69_3';
ST03_4x2_B69_3.sInit.BitName		:='+8_4x2_B69.3';
ST03_4x2_B69_3.sInit.Description	:='Zuführung Stopper AST';
ST03_4x2_B69_3.sInit.SensorType		:=sValveSensorType_WORK;

(* Init ST03_4x2_B69_4 Zuführung Stopper AST ausgefahren (ValveSensor) *)
ST03_4x2_B69_4.sInit.InstName		:='ST03_4x2_B69_4';
ST03_4x2_B69_4.sInit.BitName		:='+8_4x2_B69.4';
ST03_4x2_B69_4.sInit.Description	:='Zuführung Stopper GST';
ST03_4x2_B69_4.sInit.SensorType		:=sValveSensorType_INIT;

(* Init ST03_4x2_B69_5 ISK anwesend am Stopper (DigIn) *)
ST03_4x2_B69_5.sInit.InstName            :='ST03_4x2_B69_5';
ST03_4x2_B69_5.sInit.Description         :='ISK anwesend am Stopper';
ST03_4x2_B69_5.sInit.BitInName           :='+8-4x2_B69.5';
ST03_4x2_B69_5.sInit.HomePosSignal       :=2; (* 0: Signal=Low, 1: Signal=High, 2: always  *)
ST03_4x2_B69_5.sInit.MaxTime             :=2000;
ST03_4x2_B69_5.sInit.EnableInEveryMode   :=TRUE;

(* Init ST03_4x2_B69_6 Zuführung Stopper GST eingefahren (ValveSensor) *)
ST03_4x2_B69_6.sInit.InstName		:='ST03_4x2_B69_6';
ST03_4x2_B69_6.sInit.BitName		:='+8_4x2_B69.6';
ST03_4x2_B69_6.sInit.Description	:='Zuführung Stopper Übergabeposition AST';
ST03_4x2_B69_6.sInit.SensorType		:=sValveSensorType_WORK;

(* Init ST03_4x2_B69_7 Zuführung Stopper AST ausgefahren (ValveSensor) *)
ST03_4x2_B69_7.sInit.InstName		:='ST03_4x2_B69_7';
ST03_4x2_B69_7.sInit.BitName		:='+8_4x2_B69.7';
ST03_4x2_B69_7.sInit.Description	:='Zuführung Stopper Übergabeposition GST';
ST03_4x2_B69_7.sInit.SensorType		:=sValveSensorType_INIT;

(* Init ST03_4x3_B70_0 ISK anwesend Übergabeposition Stopper (DigIn) *)
ST03_4x3_B70_0.sInit.InstName            :='ST03_4x3_B70_0';
ST03_4x3_B70_0.sInit.Description         :='ISK anwesend Übergabeposition Stopper';
ST03_4x3_B70_0.sInit.BitInName           :='+8-4x3_B70.0';
ST03_4x3_B70_0.sInit.HomePosSignal       :=2; (* 0: Signal=Low, 1: Signal=High, 2: always  *)
ST03_4x3_B70_0.sInit.MaxTime             :=2000;
ST03_4x3_B70_0.sInit.EnableInEveryMode   :=TRUE;

(* Init ST03_4x3_B70_1 ISK anwesend Übergabeposition (DigIn) *)
ST03_4x3_B70_1.sInit.InstName            :='ST03_4x3_B70_1';
ST03_4x3_B70_1.sInit.Description         :='ISK anwesend Übergabeposition';
ST03_4x3_B70_1.sInit.BitInName           :='+8-4x3_B70.1';
ST03_4x3_B70_1.sInit.HomePosSignal       :=2; (* 0: Signal=Low, 1: Signal=High, 2: always  *)
ST03_4x3_B70_1.sInit.MaxTime             :=2000;
ST03_4x3_B70_1.sInit.EnableInEveryMode   :=TRUE;

(* Init ST03_4x3_Y70_5  Zuführung Vereinzler AST/GST (Valve) *)
ST03_4x3_Y70_5.sInit.InstName            :='ST03_4x3_Y70_5';
ST03_4x3_Y70_5.sInit.BitName            :='+8-4x3_Y70.5';
ST03_4x3_Y70_5.sInit.Description         :='Zuführung Vereinzler AST/GST';
ST03_4x3_Y70_5.sInit.HomePosDefine       :=HOME_ALWAYS;
ST03_4x3_Y70_5.sInit.InitDescription     :='GS einfahren';
ST03_4x3_Y70_5.sInit.WorkDescription     :='AS ausfahren';
ST03_4x3_Y70_5.sInit.DampBothTime        :=200;
ST03_4x3_Y70_5.sInit.KindOfValve         :='A';
ST03_4x3_Y70_5.sInit.MaxTime             :=2000;

(* Init ST03_4x3_Y70_6   Zuführung Stopper AST/GST (Valve) *)
ST03_4x3_Y70_6.sInit.InstName            :='ST03_4x3_Y70_6';
ST03_4x3_Y70_6.sInit.BitName            :='+8-4x3_Y70.6';
ST03_4x3_Y70_6.sInit.Description         :=' Zuführung Stopper AST/GST';
ST03_4x3_Y70_6.sInit.HomePosDefine       :=HOME_ALWAYS;
ST03_4x3_Y70_6.sInit.InitDescription     :='GS ausfahren';
ST03_4x3_Y70_6.sInit.WorkDescription     :='AS einfahren';
ST03_4x3_Y70_6.sInit.DampBothTime        :=200;
ST03_4x3_Y70_6.sInit.KindOfValve         :='A';
ST03_4x3_Y70_6.sInit.MaxTime             :=2000;

(* Init ST03_4x3_Y70_7   Zuführung Stopper Übergabeposition AST/GST (Valve) *)
ST03_4x3_Y70_7.sInit.InstName            :='ST03_4x3_Y70_7';
ST03_4x3_Y70_7.sInit.BitName            :='+8-4x3_Y70.7';
ST03_4x3_Y70_7.sInit.Description         :=' Zuführung Stopper Übergabeposition AST/GST';
ST03_4x3_Y70_7.sInit.HomePosDefine       :=HOME_ALWAYS;
ST03_4x3_Y70_7.sInit.InitDescription     :='GS ausfahren';
ST03_4x3_Y70_7.sInit.WorkDescription     :='AS einfahren';
ST03_4x3_Y70_7.sInit.DampBothTime        :=200;
ST03_4x3_Y70_7.sInit.KindOfValve         :='A';
ST03_4x3_Y70_7.sInit.MaxTime             :=2000;
END_ACTION

(* POU Stations/ST_08_Palettierer/ST_08__InitFBs/ST08_Init, ST *)
PROGRAM ST08_Init


VAR


END_VAR
(* ----------------------------------------------------------------------------------------- *)
(*Init ST08_180_M1 Abstapeln*)
ST08_180_M1.sConfig.Description			:='Abstapeln';
ST08_180_M1.sConfig.InstName			:='ST08_180_M1';
ST08_180_M1.sConfig.Skalierfaktor		:=360.0 / (EXPT(2,20))	; (*360°/ 20 bit Encoder =0.00034332275390625*)
ST08_180_M1.sConfig.Getriebefaktor		:=10;
ST08_180_M1.sConfig.Modulo				:=FALSE;
ST08_180_M1.sConfig.Pos_Faktor			:=5;				(*Weg bei einer Umdrehung in mm (nach Getriebe)*)
ST08_180_M1.sConfig.maxRpm				:=3500;
ST08_180_M1.sConfig.ModeOfOperation		:=CSP;			(*CSP,CSV,CST,CSTCA muss an der KLemme (Coe-Online 7010.03) eingestellt werden*)
(*(CSP) position mode*)
ST08_180_M1.sConfig.Torque_Limit		:=0;			(*bei 0 ausgeschaltet*)
ST08_180_M1.sConfig.SW_Limit_on			:=TRUE;
ST08_180_M1.sConfig.SW_Limit_min		:=-8;
ST08_180_M1.sConfig.SW_Limit_max		:=185;
ST08_180_M1.sConfig.lr_kp 				:= 800;
ST08_180_M1.sConfig.lr_ki 				:= 100.0;
ST08_180_M1.sConfig.lr_kd 				:= 50;
(* ----------------------------------------------------------------------------------------- *)
(*Init ST08_185_M1 Aufstapeln*)
ST08_185_M1.sConfig.Description		:='Aufstapeln';
ST08_185_M1.sConfig.InstName			:='ST08_185_M1';
ST08_185_M1.sConfig.Skalierfaktor		:=360.0 / (EXPT(2,20))	; (*360°/ 20 bit Encoder =0.00034332275390625*)
ST08_185_M1.sConfig.Getriebefaktor		:=10;
ST08_185_M1.sConfig.Modulo			:=FALSE;
ST08_185_M1.sConfig.Pos_Faktor		:=5;			(*Weg bei einer Umdrehung in mm (nach Getriebe)*)
ST08_185_M1.sConfig.maxRpm			:=3500;
ST08_185_M1.sConfig.ModeOfOperation	:=CSP;		(*CSP,CSV,CST,CSTCA muss an der KLemme (Coe-Online 7010.03) eingestellt werden*)
(*(CSP) position mode*)
ST08_185_M1.sConfig.Torque_Limit		:=0;			(*bei 0 ausgeschaltet*)
ST08_185_M1.sConfig.SW_Limit_on		:=TRUE;
ST08_185_M1.sConfig.SW_Limit_min		:=-8;
ST08_185_M1.sConfig.SW_Limit_max	:=185;
ST08_185_M1.sConfig.lr_kp 				:= 800;
ST08_185_M1.sConfig.lr_ki 				:= 100.0;
ST08_185_M1.sConfig.lr_kd 				:= 50;
(* ----------------------------------------------------------------------------------------- *)
(*Init ST08_190_M1 Tray ausheben*)
ST08_190_M1.sConfig.Description		:='Tray ausheben';
ST08_190_M1.sConfig.InstName			:='ST08_190_M1';
ST08_190_M1.sConfig.Skalierfaktor		:=360.0 / (EXPT(2,20))	; (*360°/ 20 bit Encoder =0.00034332275390625*)
ST08_190_M1.sConfig.Getriebefaktor		:=1;
ST08_190_M1.sConfig.Modulo			:=FALSE;
ST08_190_M1.sConfig.Pos_Faktor		:=5;			(*Weg bei einer Umdrehung in mm (nach Getriebe)*)
ST08_190_M1.sConfig.maxRpm			:=3500;
ST08_190_M1.sConfig.ModeOfOperation	:=CSP;		(*CSP,CSV,CST,CSTCA muss an der KLemme (Coe-Online 7010.03) eingestellt werden*)
(*(CSP) position mode*)
ST08_190_M1.sConfig.Torque_Limit		:=0;			(*bei 0 ausgeschaltet*)
ST08_190_M1.sConfig.SW_Limit_on		:=TRUE;
ST08_190_M1.sConfig.SW_Limit_min		:=-20;
ST08_190_M1.sConfig.SW_Limit_max	:=185;
ST08_190_M1.sConfig.lr_kp 				:= 800;
ST08_190_M1.sConfig.lr_ki 				:= 100.0;
ST08_190_M1.sConfig.lr_kd 				:= 50;
(* ----------------------------------------------------------------------------------------- *)

(* Init ST08_400_B50_0 Traystapel vor Vereinzeler Einlaufband hinten (DigIn) *)
ST08_400_B50_0.sInit.InstName            :='ST08_400_B50_0';
ST08_400_B50_0.sInit.Description         :='Traystapel hinten vor Vereinzeler Einlaufband hinten';
ST08_400_B50_0.sInit.BitInName           :='+8-400_B50.0';
ST08_400_B50_0.sInit.HomePosSignal       :=2; (* 0: Signal=Low, 1: Signal=High, 2: always  *)
ST08_400_B50_0.sInit.MaxTime             :=2000;

(* Init ST08_400_B50_4 Stopper Traystapel Einlaufband hinten rechts GST (ValveSensor) *)
ST08_400_B50_4.sInit.InstName            :='ST08_400_B50_4';
ST08_400_B50_4.sInit.BitName            :='+8_400_B50.4';
ST08_400_B50_4.sInit.Description         :='Stopper Traystapel Einlaufband hinten rechts GST';
ST08_400_B50_4.sInit.SensorType          :=sValveSensorType_INIT;

(* Init ST08_401_B50_5 Traystapel vor Vereinzeler Einlaufband mitte (DigIn) *)
ST08_401_B50_5.sInit.InstName            :='ST08_401_B50_5';
ST08_401_B50_5.sInit.Description         :='Traystapel mitte vor Vereinzeler Einlaufband ';
ST08_401_B50_5.sInit.BitInName           :='+8-401_B50.5';
ST08_401_B50_5.sInit.HomePosSignal       :=2; (* 0: Signal=Low, 1: Signal=High, 2: always  *)
ST08_401_B50_5.sInit.MaxTime             :=2000;

(* Init ST08_401_B51_1 Stopper Traystapel Einlaufband mitte rechts GST (ValveSensor) *)
ST08_401_B51_1.sInit.InstName            :='ST08_401_B51_1';
ST08_401_B51_1.sInit.BitName            :='+8_401_B51.1';
ST08_401_B51_1.sInit.Description         :='Stopper Traystapel Einlaufband mitte rechts GST';
ST08_401_B51_1.sInit.SensorType          :=sValveSensorType_INIT;


(* Init ST08_402_B51_2 Traystapel vor Vereinzeler Einlaufband vorne (DigIn) *)
ST08_402_B51_2.sInit.InstName            :='ST08_402_B51_2';
ST08_402_B51_2.sInit.Description         :='Traystapel vorne vor Vereinzeler Einlaufband ';
ST08_402_B51_2.sInit.BitInName           :='+8-402_B51.2';
ST08_402_B51_2.sInit.HomePosSignal       :=2; (* 0: Signal=Low, 1: Signal=High, 2: always  *)
ST08_402_B51_2.sInit.MaxTime             :=2000;

(*ST08_402_B51_3 Traystapel schieben mitte ausgefahren (ValveSensor)*)
ST08_402_B51_3.sInit.InstName            :='ST08_402_B51_3';
ST08_402_B51_3.sInit.BitName            :='+8_402_B51.3';
ST08_402_B51_3.sInit.Description         :='Traystapel schieben mitte';
ST08_402_B51_3.sInit.SensorType          :=sValveSensorType_INIT;

(* Init ST08_402_B51_4 (* Luftzone 1 *) (DigIn) *)
ST08_402_B51_4.sInit.InstName            :='ST08_402_B51_4';
ST08_402_B51_4.sInit.Description         :='Druckschalter St08 Zone2';
ST08_402_B51_4.sInit.BitInName           :='+8-402_B51.4';
ST08_402_B51_4.sInit.HomePosSignal       :=2; (* 0: Signal=Low, 1: Signal=High, 2: always  *)
ST08_402_B51_4.sInit.MaxTime             :=2000;
ST08_402_B51_4.sInit.EnableInEveryMode   :=TRUE;

(* Init ST08_402_B51_5 (* Luftzone 1 *) (DigIn) *)
ST08_402_B51_5.sInit.InstName            :='ST08_402_B51_5';
ST08_402_B51_5.sInit.Description         :='Druckschalter St08 Zone3';
ST08_402_B51_5.sInit.BitInName           :='+8-402_B51.5';
ST08_402_B51_5.sInit.HomePosSignal       :=2; (* 0: Signal=Low, 1: Signal=High, 2: always  *)
ST08_402_B51_5.sInit.MaxTime             :=2000;
ST08_402_B51_5.sInit.EnableInEveryMode   :=TRUE;

(* Init ST08_402_B51_6 Stopper Traystapel Einlaufband vorne rechts GST (ValveSensor) *)
ST08_402_B51_6.sInit.InstName            :='ST08_402_B51_6';
ST08_402_B51_6.sInit.BitName            :='+8_402_B51.6';
ST08_402_B51_6.sInit.Description         :='Stopper Traystapel Einlaufband vorne rechts GST';
ST08_402_B51_6.sInit.SensorType          :=sValveSensorType_INIT;

(*ST08_402_B51_7 Traystapel schieben vorne ausgefahren (ValveSensor)*)
ST08_402_B51_7.sInit.InstName            :='ST08_402_B51_7';
ST08_402_B51_7.sInit.BitName            :='+8_402_B51.7';
ST08_402_B51_7.sInit.Description         :='Traystapel schieben vorne';
ST08_402_B51_7.sInit.SensorType          :=sValveSensorType_INIT;

(* Init ST08_403_B52_0 Hubstüre 1 AST (ValveSensor) *)
ST08_403_B52_0.sInit.InstName            :='ST08_403_B52_0';
ST08_403_B52_0.sInit.BitName            :='+8_403_B52_0';
ST08_403_B52_0.sInit.Description         :='Hubtüre 1 Einlauf STN8 AST';
ST08_403_B52_0.sInit.SensorType          :=sValveSensorType_WORK;

(* Init ST08_403_B52_1 Hubstüre 1 GST  (ValveSensor) *)
ST08_403_B52_1.sInit.InstName            :='ST08_403_B52_1';
ST08_403_B52_1.sInit.BitName            :='+8_403_B52_1';
ST08_403_B52_1.sInit.Description         :='Hubtüre 1 Einlauf STN8 AST';
ST08_403_B52_1.sInit.SensorType          :=sValveSensorType_INIT;

(* Init ST08_404_B52_2 Traystapel in Ablageposition Isokörper (DigIn) *)
ST08_404_B52_2.sInit.InstName            :='ST08_404_B52_2';
ST08_404_B52_2.sInit.Description         :='Traystapel in Ablageposition Isokörper';
ST08_404_B52_2.sInit.BitInName           :='+8-404_B52.2'; 
ST08_404_B52_2.sInit.HomePosSignal       :=2; (* 0: Signal=Low, 1: Signal=High, 2: always  *)
ST08_404_B52_2.sInit.MaxTime             :=2000;

(* Init ST08_404_B52_3 Traystapel richtig eingelegt Isokörper (DigIn) *)
ST08_404_B52_3.sInit.InstName            :='ST08_404_B52_3';
ST08_404_B52_3.sInit.Description         :='Traystapel richtig eingelegt Isokörper';
ST08_404_B52_3.sInit.BitInName           :='+8-404_B52.3';
ST08_404_B52_3.sInit.HomePosSignal       :=2; (* 0: Signal=Low, 1: Signal=High, 2: always  *)
ST08_404_B52_3.sInit.MaxTime             :=2000;

(* Init ST08_406_B54_0 Tray in Zwischenp. Entnahme Isokörper (Bandende) (DigIn) *)
ST08_406_B54_0.sInit.InstName            :='ST08_406_B54_0';
ST08_406_B54_0.sInit.Description         :='Tray in Zwischenp. Entnahme Isokörper (Bandende)';
ST08_406_B54_0.sInit.BitInName           :='+8-406_B54.0';
ST08_406_B54_0.sInit.HomePosSignal       :=2; (* 0: Signal=Low, 1: Signal=High, 2: always  *)
ST08_406_B54_0.sInit.MaxTime             :=2000;

(* Init ST08_406_B54_3 Ausheber Trays in Entnahmepos.  (DigIn) *)
ST08_406_B54_3.sInit.InstName            :='ST08_406_B54_3';
ST08_406_B54_3.sInit.Description         :='Ausheber Trays in Entnahmepos. STN8 ';
ST08_406_B54_3.sInit.BitInName           :='+8-406_B54.3';
ST08_406_B54_3.sInit.HomePosSignal       :=2; (* 0: Signal=Low, 1: Signal=High, 2: always  *)
ST08_406_B54_3.sInit.MaxTime             :=2000;

(* Init ST08_406_B54_6 Ausheber Trays in Entnahmepos.  (DigIn) *)
ST08_406_B54_6.sInit.InstName            :='ST08_406_B54_6';
ST08_406_B54_6.sInit.Description         :='Tray aus Entnahmepos. ausgelaufen STN8 ';
ST08_406_B54_6.sInit.BitInName           :='+8-406_B54.6';
ST08_406_B54_6.sInit.HomePosSignal       :=2; (* 0: Signal=Low, 1: Signal=High, 2: always  *)
ST08_406_B54_6.sInit.MaxTime             :=5000;


(* Init ST08_407_B55_4 Tray in Aufstapelposition eingelaufen STN8 (DigIn) *)
ST08_407_B55_4.sInit.InstName            :='ST08_407_B55_4';
ST08_407_B55_4.sInit.Description         :='Tray in Aufstapelposition eingelaufen STN8';
ST08_407_B55_4.sInit.BitInName           :='+8-407_B55.4'; 
ST08_407_B55_4.sInit.HomePosSignal       :=2; (* 0: Signal=Low, 1: Signal=High, 2: always  *)
ST08_407_B55_4.sInit.MaxTime             :=2000;

(* Init ST08_409_B55_5 Auslaufrollenbahn voll STN8 (DigIn) *) 
ST08_409_B55_5.sInit.InstName            :='ST08_409_B55_5';
ST08_409_B55_5.sInit.Description         :='Auslaufrollenbahn voll STN8';
ST08_409_B55_5.sInit.BitInName           :='+8-409_B55.5';
ST08_409_B55_5.sInit.HomePosSignal       :=2; (* 0: Signal=Low, 1: Signal=High, 2: always  *)
ST08_409_B55_5.sInit.MaxTime             :=2000;

(* Init ST08_404_B52_4 Stopper Traystapel Isokörper AST (ValveSensor) *)
ST08_404_B52_4.sInit.InstName            :='ST08_404_B52_4';
ST08_404_B52_4.sInit.BitName            :='+8_404_B52_4';
ST08_404_B52_4.sInit.Description         :='Stopper Traystapel Isokörper AST';
ST08_404_B52_4.sInit.SensorType          :=sValveSensorType_WORK;

(* Init ST08_404_B52_5 Stopper Traystapel Isokörper GST (ValveSensor) *)
ST08_404_B52_5.sInit.InstName            :='ST08_404_B52_5';
ST08_404_B52_5.sInit.BitName            :='+8_404_B52.5';
ST08_404_B52_5.sInit.Description         :='Stopper Traystapel Isokörper GST';
ST08_404_B52_5.sInit.SensorType          :=sValveSensorType_INIT;

(* Init ST08_404_B52_6 Abstapelzylinder 1 Isokörper AST (ValveSensor) *)
ST08_404_B52_6.sInit.InstName            :='ST08_404_B52_6';
ST08_404_B52_6.sInit.BitName            :='+8_404_B52.6';
ST08_404_B52_6.sInit.Description         :='Abstapelzylinder 1 Isokörper AST';
ST08_404_B52_6.sInit.SensorType          :=sValveSensorType_WORK;

(* Init ST08_404_B52_7 Abstapelzylinder 1 Isokörper GST (ValveSensor) *)
ST08_404_B52_7.sInit.InstName            :='ST08_404_B52_7';
ST08_404_B52_7.sInit.BitName            :='+8_404_B52.7';
ST08_404_B52_7.sInit.Description         :='Abstapelzylinder 1 Isokörper GST';
ST08_404_B52_7.sInit.SensorType          :=sValveSensorType_INIT;

(* Init ST08_404_B53_0 Abstapelzylinder 2 Isokörper AST (ValveSensor) *)
ST08_404_B53_0.sInit.InstName            :='ST08_404_B53_0';
ST08_404_B53_0.sInit.BitName            :='+8_404_B53.0';
ST08_404_B53_0.sInit.Description         :='Abstapelzylinder 2 Isokörper AST';
ST08_404_B53_0.sInit.SensorType          :=sValveSensorType_WORK;

(* Init ST08_404_B53_1 Abstapelzylinder 2 Isokörper GST (ValveSensor) *)
ST08_404_B53_1.sInit.InstName            :='ST08_404_B53_1';
ST08_404_B53_1.sInit.BitName            :='+8_404_B53.1';
ST08_404_B53_1.sInit.Description         :='Abstapelzylinder 2 Isokörper GST';
ST08_404_B53_1.sInit.SensorType          :=sValveSensorType_INIT;

(* Init ST08_405_B53_2 Rückhaltezylinder links Traystapel Isokörper AST (ValveSensor) *)
ST08_405_B53_2.sInit.InstName            :='ST08_405_B53_2';
ST08_405_B53_2.sInit.BitName            :='+8_405_B53.2';
ST08_405_B53_2.sInit.Description         :='Rückhaltezylinder links Traystapel Isokörper AST';
ST08_405_B53_2.sInit.SensorType          :=sValveSensorType_WORK;

(* Init ST08_405_B53_3 Rückhaltezylinder links Traystapel Isokörper GST (ValveSensor) *)
ST08_405_B53_3.sInit.InstName            :='ST08_405_B53_3';
ST08_405_B53_3.sInit.BitName            :='+8_405_B53.3';
ST08_405_B53_3.sInit.Description         :='Rückhaltezylinder links Traystapel Isokörper GST';
ST08_405_B53_3.sInit.SensorType          :=sValveSensorType_INIT;

(* Init ST08_405_B53_4 Rückhaltezylinder rechts Traystapel Isokörper AST (ValveSensor) *)
ST08_405_B53_4.sInit.InstName            :='ST08_405_B53_4';
ST08_405_B53_4.sInit.BitName            :='+8_405_B53.4';
ST08_405_B53_4.sInit.Description         :='Rückhaltezylinder rechts Traystapel Isokörper AST';
ST08_405_B53_4.sInit.SensorType          :=sValveSensorType_WORK;

(* Init ST08_405_B53_5 Rückhaltezylinder rechts Traystapel Isokörper GST (ValveSensor) *)
ST08_405_B53_5.sInit.InstName            :='ST08_405_B53_5';
ST08_405_B53_5.sInit.BitName            :='+8_405_B53.5';
ST08_405_B53_5.sInit.Description         :='Rückhaltezylinder rechts Traystapel Isokörper GST';
ST08_405_B53_5.sInit.SensorType          :=sValveSensorType_INIT;

(* Init ST08_405_B53_6 Hubtüre 2 Einlauf Isokörper STN8 AST (ValveSensor) *)
ST08_405_B53_6.sInit.InstName            :='ST08_405_B53_6';
ST08_405_B53_6.sInit.BitName            :='+8_405_B53.6';
ST08_405_B53_6.sInit.Description         :='Hubtüre 2 Einlauf Isokörper STN8 AST';
ST08_405_B53_6.sInit.SensorType          :=sValveSensorType_WORK;

(* Init ST08_405_B53_7 Hubtüre 2 Einlauf Isokörper STN8 GST (ValveSensor) *)
ST08_405_B53_7.sInit.InstName            :='ST08_405_B53_7';
ST08_405_B53_7.sInit.BitName            :='+8_405_B53.7';
ST08_405_B53_7.sInit.Description         :='Hubtüre 2 Einlauf Isokörper STN8 GST';
ST08_405_B53_7.sInit.SensorType          :=sValveSensorType_Init;

(* Init ST08_406_B54_1 Hub Bandstrecke 2und 3 STN8 AST (ValveSensor) *)
ST08_406_B54_1.sInit.InstName            :='ST08_406_B54_1';
ST08_406_B54_1.sInit.BitName            :='+8_406_B54.1';
ST08_406_B54_1.sInit.Description         :='Hub Bandstrecke 2 und 3 STN8 AST';
ST08_406_B54_1.sInit.SensorType          :=sValveSensorType_WORK;

(* Init ST08_406_B54_2 Hub Bandstrecke 2und 3 STN8 GST (ValveSensor) *)
ST08_406_B54_2.sInit.InstName            :='ST08_406_B54_2';
ST08_406_B54_2.sInit.BitName            :='+8_406_B54.2';
ST08_406_B54_2.sInit.Description         :='Hub Bandstrecke 2und 3 STN8 GST';
ST08_406_B54_2.sInit.SensorType          :=sValveSensorType_INIT;

(* Init ST08_406_B54_4 Ausheber Trays Entnahmepos. Isok. STN8 GST (ValveSensor) *)
ST08_406_B54_4.sInit.InstName            :='ST08_406_B54';
ST08_406_B54_4.sInit.BitName            :='+8_406_B54.4';
ST08_406_B54_4.sInit.Description         :='Ausheber Trays Entnahmepos. Isok. STN8 AST';
ST08_406_B54_4.sInit.SensorType          :=sValveSensorType_WORK;

(* Init ST08_406_B54_4 Ausheber Trays Entnahmepos. Isok. STN8 GST (ValveSensor) *)
ST08_406_B54_5.sInit.InstName            :='ST08_406_B54_5';
ST08_406_B54_5.sInit.BitName            :='+8_406_B54.5';
ST08_406_B54_5.sInit.Description         :='Ausheber Trays Entnahmepos. Isok. STN8 GST';
ST08_406_B54_5.sInit.SensorType          :=sValveSensorType_INIT;

(* Init ST08_407_B55_0 Hubtüre 3 Auslauf STN8 AST (ValveSensor) *)
ST08_407_B55_0.sInit.InstName            :='ST08_407_B55_0';
ST08_407_B55_0.sInit.BitName            :='+8_407_B55.0';
ST08_407_B55_0.sInit.Description         :='Hubtüre 3 Auslauf STN8 AST';
ST08_407_B55_0.sInit.SensorType          :=sValveSensorType_WORK;

(* Init ST08_407_B55_1 Hubtüre 3 Auslauf STN8 AST (ValveSensor) *)
ST08_407_B55_1.sInit.InstName            :='ST08_407_B55_1';
ST08_407_B55_1.sInit.BitName            :='+8_407_B55.1';
ST08_407_B55_1.sInit.Description         :='Hubtüre 3 Auslauf STN8 GST';
ST08_407_B55_1.sInit.SensorType          :=sValveSensorType_INIT;

(* Init ST08_407_B55_2 Hubtüre 4 Auslauf STN8 AST (ValveSensor) *)
ST08_407_B55_2.sInit.InstName            :='ST08_407_B55_2';
ST08_407_B55_2.sInit.BitName            :='+8_407_B55.2';
ST08_407_B55_2.sInit.Description         :='Hubtüre 4 Auslauf STN8 AST';
ST08_407_B55_2.sInit.SensorType          :=sValveSensorType_WORK;

(* Init ST08_407_B55_3 Hubtüre 4 Auslauf STN8 AST (ValveSensor) *)
ST08_407_B55_3.sInit.InstName            :='ST08_407_B55_3';
ST08_407_B55_3.sInit.BitName            :='+8_407_B55.3';
ST08_407_B55_3.sInit.Description         :='Hubtüre 4 Auslauf STN8 GST';
ST08_407_B55_3.sInit.SensorType          :=sValveSensorType_INIT;

(* Init ST08_408_B56_0 Rückhaltezylinder links Auslauf STN8 AST (ValveSensor) *)
ST08_408_B56_0.sInit.InstName            :='ST08_408_B56_0';
ST08_408_B56_0.sInit.BitName            :='+8_408_B56.0';
ST08_408_B56_0.sInit.Description         :='Rückhaltezylinder links Auslauf STN8 AST';
ST08_408_B56_0.sInit.SensorType          :=sValveSensorType_WORK;

(* Init ST08_408_B56_1 Rückhaltezylinder links Auslauf STN8 GST (ValveSensor) *)
ST08_408_B56_1.sInit.InstName            :='ST08_408_B56_1';
ST08_408_B56_1.sInit.BitName            :='+8_408_B56.1';
ST08_408_B56_1.sInit.Description         :='Rückhaltezylinder links Auslauf STN8 GST';
ST08_408_B56_1.sInit.SensorType          :=sValveSensorType_INIT;

(* Init ST08_408_B56_2 Rückhaltezylinder rechts Auslauf STN8 AST (ValveSensor) *)
ST08_408_B56_2.sInit.InstName            :='ST08_408_B56_2';
ST08_408_B56_2.sInit.BitName            :='+8_408_B56.2';
ST08_408_B56_2.sInit.Description         :='Rückhaltezylinder rechts Auslauf STN8 AST';
ST08_408_B56_2.sInit.SensorType          :=sValveSensorType_WORK;

(* Init ST08_408_B56_3 Rückhaltezylinder rechts Auslauf STN8 GST (ValveSensor) *)
ST08_408_B56_3.sInit.InstName            :='ST08_408_B56_3';
ST08_408_B56_3.sInit.BitName            :='+8_408_B56.3';
ST08_408_B56_3.sInit.Description         :='Rückhaltezylinder rechts Auslauf STN8 GST';
ST08_408_B56_3.sInit.SensorType          :=sValveSensorType_INIT;

(* Init ST08_408_B56_4 Abstapelzylinder 1 STN8 AST (ValveSensor) *)
ST08_408_B56_4.sInit.InstName            :='ST08_408_B56_4';
ST08_408_B56_4.sInit.BitName            :='+8_408_B56.4';
ST08_408_B56_4.sInit.Description         :='Abstapelzylinder 1 STN8 AST';
ST08_408_B56_4.sInit.SensorType          :=sValveSensorType_WORK;

(* Init ST08_408_B56_5 Abstapelzylinder 1 STN8 GST (ValveSensor) *)
ST08_408_B56_5.sInit.InstName            :='ST08_408_B56_5';
ST08_408_B56_5.sInit.BitName            :='+8_408_B56.5';
ST08_408_B56_5.sInit.Description         :='Abstapelzylinder 1 STN8 GST';
ST08_408_B56_5.sInit.SensorType          :=sValveSensorType_INIT;

(* Init ST08_408_B56_6 Abstapelzylinder 2 STN8 AST (ValveSensor) *)
ST08_408_B56_6.sInit.InstName            :='ST08_408_B56_6';
ST08_408_B56_6.sInit.BitName            :='+8_408_B56.6';
ST08_408_B56_6.sInit.Description         :='Abstapelzylinder 2 STN8 AST';
ST08_408_B56_6.sInit.SensorType          :=sValveSensorType_WORK;

(* Init ST08_408_B56_7 Abstapelzylinder 2 STN8 AST (ValveSensor) *)
ST08_408_B56_7.sInit.InstName            :='ST08_408_B56_7';
ST08_408_B56_7.sInit.BitName            :='+8_408_B56.7';
ST08_408_B56_7.sInit.Description         :='Abstapelzylinder 2 STN8 GST';
ST08_408_B56_7.sInit.SensorType          :=sValveSensorType_INIT;

(*ST08_400_B50_1 Stopper links + rechts Traystapel Auslaufband eingefahren (ValveSensor)*)
ST08_400_B50_1.sInit.InstName            :='ST08_400_B50_1';
ST08_400_B50_1.sInit.BitName            :='+8_400_B50.1';
ST08_400_B50_1.sInit.Description         :='Stopper links + rechts Auslauf STN8 AST';
ST08_400_B50_1.sInit.SensorType          :=sValveSensorType_WORK;

(*ST08_400_B50_2 Stopper links + rechts Traystapel Auslaufband ausgefahren (ValveSensor)*)
ST08_400_B50_2.sInit.InstName            :='ST08_400_B50_2';
ST08_400_B50_2.sInit.BitName            :='+8_400_B50.2';
ST08_400_B50_2.sInit.Description         :='Stopper links + rechts Auslauf STN8 GST';
ST08_400_B50_2.sInit.SensorType          :=sValveSensorType_INIT;

(*ST08_400_B50_3 Stopper links + rechts Traystapel Auslaufband eingefahren (ValveSensor)*)
ST08_400_B50_3.sInit.InstName            :='ST08_400_B50_3';
ST08_400_B50_3.sInit.BitName            :='+8_400_B50.3';
ST08_400_B50_3.sInit.Description         :='Stopper links + rechts Auslauf STN8 AST';
ST08_400_B50_3.sInit.SensorType          :=sValveSensorType_WORK;

(*ST08_400_B50_6 Stopper links + rechts Traystapel Auslaufband ausgefahren (ValveSensor)*)
ST08_400_B50_6.sInit.InstName            :='ST08_400_B50_6';
ST08_400_B50_6.sInit.BitName            :='+8_400_B50.6';
ST08_400_B50_6.sInit.Description         :='Stopper links + rechts Auslauf STN8 GST';
ST08_400_B50_6.sInit.SensorType          :=sValveSensorType_INIT;

(*ST08_401_B50_7 Traystapel schieben hinten ausgefahren (ValveSensor)*)
ST08_401_B50_7.sInit.InstName            :='ST08_401_B50_7';
ST08_401_B50_7.sInit.BitName            :='+8_401_B50.7';
ST08_401_B50_7.sInit.Description         :='Traystapel schieben hinten';
ST08_401_B50_7.sInit.SensorType          :=sValveSensorType_INIT;

(*ST08_412_B58_0 Rüstsatz Förderband Vereinzelner ausgefahren (ValveSensor)*)
ST08_412_B58_0.sInit.InstName            :='ST08_412_B58_0';
ST08_412_B58_0.sInit.BitName          	 :='+8_412_B58.0';
ST08_412_B58_0.sInit.Description         :='Rüstsatz Förderband Vereinzelner STN8 AST';
ST08_412_B58_0.sInit.SensorType          :=sValveSensorType_WORK;

(*ST08_412_B58_1 Rüstsatz Förderband Vereinzelner eingefahren (ValveSensor)*)
ST08_412_B58_1.sInit.InstName            :='ST08_412_B58_1';
ST08_412_B58_1.sInit.BitName          	 :='+8_412_B58.1';
ST08_412_B58_1.sInit.Description         :='Rüstsatz Förderband Vereinzelner STN8 GST';
ST08_412_B58_1.sInit.SensorType          :=sValveSensorType_INIT;

(*ST08_412_B58_2 Rüstsatz Förderband Stopper ausgefahren (ValveSensor)*)
ST08_412_B58_2.sInit.InstName            :='ST08_412_B58_2';
ST08_412_B58_2.sInit.BitName           	 :='+8_412_B58.2';
ST08_412_B58_2.sInit.Description         :='Rüstsatz Förderband Stopper STN8 AST';
ST08_412_B58_2.sInit.SensorType          :=sValveSensorType_WORK;

(*ST08_412_B58_3 Rüstsatz Förderband Stopper eingefahren (ValveSensor)*)
ST08_412_B58_3.sInit.InstName            :='ST08_412_B58_3';
ST08_412_B58_3.sInit.BitName            :='+8_412_B58.3';
ST08_412_B58_3.sInit.Description         :='Rüstsatz Förderband Stopper STN8 GST';
ST08_412_B58_3.sInit.SensorType          :=sValveSensorType_INIT;

(* Init ST08_412_B58_4 Rüstsatz Förderband frei zum Ablegen ISK von SP Maschine Position 1 (DigIn) *)
ST08_412_B58_4.sInit.InstName            :='ST08_412_B58_4';
ST08_412_B58_4.sInit.Description         :='Frei SP Maschine Position 1';
ST08_412_B58_4.sInit.BitInName           :='+8-412_B58.4';
ST08_412_B58_4.sInit.HomePosSignal       :=2; (* 0: Signal=Low, 1: Signal=High, 2: always  *)
ST08_412_B58_4.sInit.MaxTime             :=2000;

(* Init ST08_412_B58_5 Rüstsatz Förderband frei zum Ablegen ISK von SP Maschine Position 2 (DigIn) *)
ST08_412_B58_5.sInit.InstName            :='ST08_412_B58_5';
ST08_412_B58_5.sInit.Description         :='Frei SP Maschine Position 2';
ST08_412_B58_5.sInit.BitInName           :='+8-412_B58.5';
ST08_412_B58_5.sInit.HomePosSignal       :=2; (* 0: Signal=Low, 1: Signal=High, 2: always  *)
ST08_412_B58_5.sInit.MaxTime             :=2000;

(* Init ST08_412_B58_6 Rüstsatz Förderband frei zum Ablegen ISK von SP Maschine Position 3 (DigIn) *)
ST08_412_B58_6.sInit.InstName            :='ST08_412_B58_6';
ST08_412_B58_6.sInit.Description         :='Frei SP Maschine Position 3';
ST08_412_B58_6.sInit.BitInName           :='+8-412_B58.6';
ST08_412_B58_6.sInit.HomePosSignal       :=2; (* 0: Signal=Low, 1: Signal=High, 2: always  *)
ST08_412_B58_6.sInit.MaxTime             :=2000;

(* Init ST08_412_B58_5_35pol Lageerkennung links (DigIn) *)
ST08_412_B58_5_35pol.sInit.InstName            :='ST08_412_B58_5_35pol';
ST08_412_B58_5_35pol.sInit.Description         :=' Lageerkennung rechts';
ST08_412_B58_5_35pol.sInit.BitInName           :='+8-412_B58.5';
ST08_412_B58_5_35pol.sInit.HomePosSignal       :=2; (* 0: Signal=Low, 1: Signal=High, 2: always  *)
ST08_412_B58_5_35pol.sInit.MaxTime             :=2000;

(* Init ST08_412_B58_6_35pol Lageerkennung rechts (DigIn) *)
ST08_412_B58_6_35pol.sInit.InstName            :='ST08_412_B58_6_35pol';
ST08_412_B58_6_35pol.sInit.Description         :=' Lageerkennung links';
ST08_412_B58_6_35pol.sInit.BitInName           :='+8-412_B58.6';
ST08_412_B58_6_35pol.sInit.HomePosSignal    :=2; (* 0: Signal=Low, 1: Signal=High, 2: always  *)
ST08_412_B58_6_35pol.sInit.MaxTime             :=2000;

(* Init ST08_412_B58_7 Rüstsatz Förderband ISK anwesend zum Vereinzeln (DigIn) *)
ST08_412_B58_7.sInit.InstName            :='ST08_412_B58_7';
ST08_412_B58_7.sInit.Description         :='ISK anwesend zum Vereinzeln';
ST08_412_B58_7.sInit.BitInName           :='+8-412_B58.7';
ST08_412_B58_7.sInit.HomePosSignal       :=2; (* 0: Signal=Low, 1: Signal=High, 2: always  *)
ST08_412_B58_7.sInit.MaxTime             :=2000;

(* Init ST08_412_B59_0 Rüstsatz Förderband ISK auf Übergabeposition Roboter Verpackung (DigIn) *)
ST08_412_B59_0.sInit.InstName            :='ST08_412_B59_0';
ST08_412_B59_0.sInit.Description         :='ISK auf Übergabeposition Roboter';
ST08_412_B59_0.sInit.BitInName           :='+8-412_B59.0';
ST08_412_B59_0.sInit.HomePosSignal       :=2; (* 0: Signal=Low, 1: Signal=High, 2: always  *)
ST08_412_B59_0.sInit.MaxTime             :=2000;

(* Init ST08_169_K1 Bandantrieb 1 Einlauf Trays Ein (DigOutIn) *)
ST08_169_K1.sInit.InstName               :='ST08_169_K1';
ST08_169_K1.sInit.Description            :='Bandantrieb 1 Einlauf Trays Ein';
ST08_169_K1.sInit.BitOutName             :='+8-169_K1'; 
ST08_169_K1.sInit.BitInName              :='';
ST08_169_K1.sInit.HomePosOutput          :=2; (* 0: Signal=Low, 1: Signal=High, 2: always  *)
ST08_169_K1.sInit.MaxTime                :=2000;
ST08_169_K1.sInit.EnableInEveryMode  :=TRUE;

(* Init ST08_169_K2 Bandantrieb 4 Auslauf leere Trays Ein (DigOutIn) *)
ST08_169_K2.sInit.InstName               :='ST08_169_K2';
ST08_169_K2.sInit.Description            :='Bandantrieb 4 Auslauf leere Trays Ein';
ST08_169_K2.sInit.BitOutName             :='+8-169_K2'; 
ST08_169_K2.sInit.BitInName              :='';
ST08_169_K2.sInit.HomePosOutput          :=2; (* 0: Signal=Low, 1: Signal=High, 2: always  *)
ST08_169_K2.sInit.MaxTime                :=2000;
ST08_169_K2.sInit.EnableInEveryMode  :=TRUE;

(* Init ST08_170_K1 Bandantrieb 2 Hubquereinheit Trays Ein (DigOutIn) *) 
ST08_170_K1.sInit.InstName               :='ST08_170_K1';
ST08_170_K1.sInit.Description            :='Bandantrieb 2 Hubquereinheit Trays Ein';
ST08_170_K1.sInit.BitOutName             :='+8-170_K1';
ST08_170_K1.sInit.BitInName              :='';
ST08_170_K1.sInit.HomePosOutput          :=2; (* 0: Signal=Low, 1: Signal=High, 2: always  *)
ST08_170_K1.sInit.MaxTime                :=2000;
ST08_170_K1.sInit.EnableInEveryMode  :=TRUE;

(* Init ST08_170_K2 Bandantrieb 3 Hubquereinheit Trays Ein (DigOutIn) *)
ST08_170_K2.sInit.InstName               :='ST08_170_K2';
ST08_170_K2.sInit.Description            :='Bandantrieb 3 Hubquereinheit Trays Ein';
ST08_170_K2.sInit.BitOutName             :='+8-170_K2';
ST08_170_K2.sInit.BitInName              :='';
ST08_170_K2.sInit.HomePosOutput          :=2; (* 0: Signal=Low, 1: Signal=High, 2: always  *)
ST08_170_K2.sInit.MaxTime                :=2000;
ST08_170_K2.sInit.EnableInEveryMode  :=TRUE;

(* Init ST08_400_Y50_0 Stopper Traystapel Einlaufb. hinten links + rechts AST (Valve) *)
ST08_400_Y50_0.sInit.InstName            :='ST08_400_Y50_0';
ST08_400_Y50_0.sInit.BitName            :='+8-400_Y50.0';
ST08_400_Y50_0.sInit.Description         :='Stopper Traystapel Einlaufb. hinten links + rechts AST';
ST08_400_Y50_0.sInit.HomePosDefine       :=HOME_INIT;
ST08_400_Y50_0.sInit.InitDescription     :='GS ausfahren';
ST08_400_Y50_0.sInit.WorkDescription     :='AS einfahren';
ST08_400_Y50_0.sInit.DampBothTime        :=200;
ST08_400_Y50_0.sInit.KindOfValve         :='2G';
ST08_400_Y50_0.sInit.MaxTime             :=2000;

(* Init ST08_400_Y50_2 Stopper Traystapel Einlaufb. mitte links + rechts AST (Valve) *)
ST08_400_Y50_2.sInit.InstName            :='ST08_400_Y50_2';
ST08_400_Y50_2.sInit.BitName            :='+8-400_Y50.2';
ST08_400_Y50_2.sInit.Description         :='Stopper Traystapel Einlaufb. mitte links + rechts AST';
ST08_400_Y50_2.sInit.HomePosDefine       :=HOME_INIT;
ST08_400_Y50_2.sInit.InitDescription     :='GS ausfahren';
ST08_400_Y50_2.sInit.WorkDescription     :='AS einfahren';
ST08_400_Y50_2.sInit.DampBothTime        :=200;
ST08_400_Y50_2.sInit.KindOfValve         :='2G';
ST08_400_Y50_2.sInit.MaxTime             :=2000;

(* Init ST08_402_Y50_4 Stopper Traystapel Einlaufb. vorne links + rechts AST (Valve) *) 
ST08_402_Y50_4.sInit.InstName            :='ST08_402_Y50_4';
ST08_402_Y50_4.sInit.BitName            :='+8-402_Y50.4';
ST08_402_Y50_4.sInit.Description         :='Stopper Traystapel Einlaufb. vorne links + rechts AST';
ST08_402_Y50_4.sInit.HomePosDefine       :=HOME_INIT;
ST08_402_Y50_4.sInit.InitDescription     :='GS ausfahren';
ST08_402_Y50_4.sInit.WorkDescription     :='AS einfahren';
ST08_402_Y50_4.sInit.DampBothTime        :=200;
ST08_402_Y50_4.sInit.KindOfValve         :='2G';
ST08_402_Y50_4.sInit.MaxTime             :=2000;

(* Init ST08_403_Y50_6 Vakuum 1 Einlauf STN8 AST (Valve) *)
ST08_403_Y50_6.sInit.InstName            :='ST08_403_Y50_6';
ST08_403_Y50_6.sInit.BitName            :='+8-403_Y50.6';
ST08_403_Y50_6.sInit.Description         :='Vakuum 1 Einlauf STN8 AST';
ST08_403_Y50_6.sInit.HomePosDefine       :=HOME_ALWAYS;
ST08_403_Y50_6.sInit.InitDescription     :='OFF';
ST08_403_Y50_6.sInit.WorkDescription     :='ON';
ST08_403_Y50_6.sInit.DampBothTime        :=0;
ST08_403_Y50_6.sInit.KindOfValve         :='A';
ST08_403_Y50_6.sInit.MaxTime             :=2000;

(* Init ST08_403_Y50_7 Vakuum 2 Einlauf STN8 AST (Valve) *)
ST08_403_Y50_7.sInit.InstName            :='ST08_403_Y50_7';
ST08_403_Y50_7.sInit.BitName            :='+8-403_Y50.7';
ST08_403_Y50_7.sInit.Description         :='Vakuum 2 Einlauf STN8 AST';
ST08_403_Y50_7.sInit.HomePosDefine       :=HOME_ALWAYS;
ST08_403_Y50_7.sInit.InitDescription     :='OFF';
ST08_403_Y50_7.sInit.WorkDescription     :='ON';
ST08_403_Y50_7.sInit.DampBothTime        :=0;
ST08_403_Y50_7.sInit.KindOfValve         :='A';
ST08_403_Y50_7.sInit.MaxTime             :=2000;

(* Init ST08_405_Y51_0 Hubtüre 2 Einlauf Isokörper STN8 AST (Valve) *)
ST08_405_Y51_0.sInit.InstName            :='ST08_405_Y51_0';
ST08_405_Y51_0.sInit.BitName            :='+8-405_Y51.0';
ST08_405_Y51_0.sInit.Description         :='Hubtüre 2 Einlauf Isokörper STN8 AST';
ST08_405_Y51_0.sInit.HomePosDefine       :=HOME_INIT;
ST08_405_Y51_0.sInit.InitDescription     :='GS ausfahren';
ST08_405_Y51_0.sInit.WorkDescription     :='AS einfahren';
ST08_405_Y51_0.sInit.DampBothTime        :=0;
ST08_405_Y51_0.sInit.KindOfValve         :='2G';
ST08_405_Y51_0.sInit.MaxTime             :=5000;

(* Init ST08_406_Y51_2 Hubtüre 3 STN8 AST (Valve) *)
ST08_406_Y51_2.sInit.InstName            :='ST08_406_Y51_2';
ST08_406_Y51_2.sInit.BitName            :='+8-406_Y51.2';
ST08_406_Y51_2.sInit.Description         :='Hubtüre 3 Auslauf STN8 AST';
ST08_406_Y51_2.sInit.HomePosDefine       :=HOME_INIT;
ST08_406_Y51_2.sInit.InitDescription     :='GS ausfahren';
ST08_406_Y51_2.sInit.WorkDescription     :='AS einfahren';
ST08_406_Y51_2.sInit.DampBothTime        :=0;
ST08_406_Y51_2.sInit.KindOfValve         :='2G';
ST08_406_Y51_2.sInit.MaxTime             :=5000;

(* Init ST08_407_Y51_4 Hubtüre 4 Auslauf STN8 AST (Valve) *)
ST08_407_Y51_4.sInit.InstName            :='ST08_407_Y51_4';
ST08_407_Y51_4.sInit.BitName            :='+8-407_Y51.4';
ST08_407_Y51_4.sInit.Description         :='Hubtüre 4 Auslauf STN8 AST';
ST08_407_Y51_4.sInit.HomePosDefine       :=HOME_ALWAYS;
ST08_407_Y51_4.sInit.InitDescription     :='GS ausfahren';
ST08_407_Y51_4.sInit.WorkDescription     :='AS einfahren';
ST08_407_Y51_4.sInit.DampBothTime        :=0;
ST08_407_Y51_4.sInit.KindOfValve         :='2G';
ST08_407_Y51_4.sInit.MaxTime             :=10000;

(* Init ST08_404_Y51_6 Stopper Traystapel Isokörper AST (Valve) *)
ST08_404_Y51_6.sInit.InstName            :='ST08_404_Y51_6';
ST08_404_Y51_6.sInit.BitName            :='+8-404_Y51.6';
ST08_404_Y51_6.sInit.Description         :='Stopper Traystapel Isokörper AST';
ST08_404_Y51_6.sInit.HomePosDefine       :=HOME_INIT;
ST08_404_Y51_6.sInit.InitDescription     :='GS ausfahren';
ST08_404_Y51_6.sInit.WorkDescription     :='AS einfahren';
ST08_404_Y51_6.sInit.DampBothTime        :=200;
ST08_404_Y51_6.sInit.KindOfValve         :='2G';
ST08_404_Y51_6.sInit.MaxTime             :=2000;

(* Init ST08_404_Y52_0 Hub Bandstrecke STN8 AST (Valve) *)
ST08_404_Y52_0.sInit.InstName            :='ST08_404_Y52_0';
ST08_404_Y52_0.sInit.BitName            :='+8-404_Y52.0';
ST08_404_Y52_0.sInit.Description         :='Hub Bandstrecke STN8 AST';
ST08_404_Y52_0.sInit.HomePosDefine       :=HOME_INIT;
ST08_404_Y52_0.sInit.InitDescription     :='GS einfahren';
ST08_404_Y52_0.sInit.WorkDescription     :='AS ausfahren';
ST08_404_Y52_0.sInit.DampBothTime        :=200;
ST08_404_Y52_0.sInit.KindOfValve         :='2G';
ST08_404_Y52_0.sInit.MaxTime             :=2000;


(* Init ST08_406_Y52_3 Ausheber Trays Entnahmepos. Isok. STN8 GST (Valve) *)
ST08_406_Y52_3.sInit.InstName            :='ST08_406_Y52_3';
ST08_406_Y52_3.sInit.BitName            :='+8-406_Y52.3';
ST08_406_Y52_3.sInit.Description         :='Ausheber Trays Entnahmepos. Isok. STN8 GST';
ST08_406_Y52_3.sInit.HomePosDefine       :=HOME_ALWAYS;
ST08_406_Y52_3.sInit.InitDescription     :='GS einfahren';
ST08_406_Y52_3.sInit.WorkDescription     :='AS ausfahren';
ST08_406_Y52_3.sInit.DampBothTime        :=200;
ST08_406_Y52_3.sInit.KindOfValve         :='2G';
ST08_406_Y52_3.sInit.MaxTime             :=3000;

(* Init ST08_401_Y52_4 Traystapel schieben hinten AST (Valve) *)
ST08_401_Y52_4.sInit.InstName            :='ST08_401_Y52_4';
ST08_401_Y52_4.sInit.BitName            :='+8-401_Y52.4';
ST08_401_Y52_4.sInit.Description         :='Traystapel schieben hinten';
ST08_401_Y52_4.sInit.HomePosDefine       :=HOME_INIT;
ST08_401_Y52_4.sInit.InitDescription     :='GS einfahren';
ST08_401_Y52_4.sInit.WorkDescription     :='AS ausfahren';
ST08_401_Y52_4.sInit.DampBothTime        :=200;
ST08_401_Y52_4.sInit.KindOfValve         :='2G';
ST08_401_Y52_4.sInit.MaxTime             :=2000;

(* Stopper links + rechts Traystapel Auslaufband einfahren (Valve) *)
ST08_400_Y52_5.sInit.InstName            :='ST08_400_Y52_5';
ST08_400_Y52_5.sInit.BitName            :='+8-400_Y52.5';
ST08_400_Y52_5.sInit.Description         :='Stopperzylinder li+re STN8 AST';
ST08_400_Y52_5.sInit.HomePosDefine       :=HOME_BOTH;
ST08_400_Y52_5.sInit.InitDescription     :='GS ausfahren';
ST08_400_Y52_5.sInit.WorkDescription     :='AS einfahren';
ST08_400_Y52_5.sInit.DampBothTime        :=200;
ST08_400_Y52_5.sInit.KindOfValve         :='2G';
ST08_400_Y52_5.sInit.MaxTime             :=3000;

(* Init ST08_402_Y52_6 Traystapel schieben mitte AST (Valve) *)
ST08_402_Y52_6.sInit.InstName            :='ST08_402_Y52_6';
ST08_402_Y52_6.sInit.BitName            :='+8-402_Y52.6';
ST08_402_Y52_6.sInit.Description         :='Traystapel schieben mitte';
ST08_402_Y52_6.sInit.HomePosDefine       :=HOME_INIT;
ST08_402_Y52_6.sInit.InitDescription     :='GS einfahren';
ST08_402_Y52_6.sInit.WorkDescription     :='AS ausfahren';
ST08_402_Y52_6.sInit.DampBothTime        :=200;
ST08_402_Y52_6.sInit.KindOfValve         :='2G';
ST08_402_Y52_6.sInit.MaxTime             :=2000;

(* Init ST08_402_Y52_7 Traystapel schieben vorne AST (Valve) *)
ST08_402_Y52_7.sInit.InstName            :='ST08_402_Y52_7';
ST08_402_Y52_7.sInit.BitName            :='+8-402_Y52.7';
ST08_402_Y52_7.sInit.Description         :='Traystapel schieben vorne';
ST08_402_Y52_7.sInit.HomePosDefine       :=HOME_INIT;
ST08_402_Y52_7.sInit.InitDescription     :='GS einfahren';
ST08_402_Y52_7.sInit.WorkDescription     :='AS ausfahren';
ST08_402_Y52_7.sInit.DampBothTime        :=200;
ST08_402_Y52_7.sInit.KindOfValve         :='2G';
ST08_402_Y52_7.sInit.MaxTime             :=2000;

(* Init ST08_404_Y53_0 Abstapelzylinder 1 AST (Valve) *)
ST08_404_Y53_0.sInit.InstName            :='ST08_404_Y53_0';
ST08_404_Y53_0.sInit.BitName            :='+8-404_Y53.0';
ST08_404_Y53_0.sInit.Description         :='Abstapelzylinder 1 AST';
ST08_404_Y53_0.sInit.HomePosDefine       :=HOME_INIT;
ST08_404_Y53_0.sInit.InitDescription     :='GS einfahren';
ST08_404_Y53_0.sInit.WorkDescription     :='AS ausfahren';
ST08_404_Y53_0.sInit.DampBothTime        :=400;
ST08_404_Y53_0.sInit.KindOfValve         :='2G';
ST08_404_Y53_0.sInit.MaxTime             :=3000;

(* Init ST08_404_Y53_2 Abstapelzylinder 2  AST (Valve) *)
ST08_404_Y53_2.sInit.InstName            :='ST08_404_Y53_2';
ST08_404_Y53_2.sInit.BitName            :='+8-404_Y53.2';
ST08_404_Y53_2.sInit.Description         :='Abstapelzylinder 2  AST';
ST08_404_Y53_2.sInit.HomePosDefine       :=HOME_INIT;
ST08_404_Y53_2.sInit.InitDescription     :='GS einfahren';
ST08_404_Y53_2.sInit.WorkDescription     :='AS ausfahren';
ST08_404_Y53_2.sInit.DampBothTime        :=200;
ST08_404_Y53_2.sInit.KindOfValve         :='2G';
ST08_404_Y53_2.sInit.MaxTime             :=3000;

(* Init ST08_405_Y53_4 Rückhaltezylinder li+re Traystapel Isokörper AST (Valve) *) 
ST08_405_Y53_4.sInit.InstName            :='ST08_405_Y53_4';
ST08_405_Y53_4.sInit.BitName            :='+8-405_Y53.4';
ST08_405_Y53_4.sInit.Description         :='Rückhaltezylinder li+re Traystapel Isokörper AST';
ST08_405_Y53_4.sInit.HomePosDefine       :=HOME_ALWAYS;
ST08_405_Y53_4.sInit.InitDescription     :='GS einfahren';
ST08_405_Y53_4.sInit.WorkDescription     :='AS ausfahren';
ST08_405_Y53_4.sInit.DampBothTime        :=200;
ST08_405_Y53_4.sInit.KindOfValve         :='2G';
ST08_405_Y53_4.sInit.MaxTime             :=3000;

(* Init ST08_408_Y54_0 Rückhaltezylinder li.+re. Auslauf STN8 AST (Valve) *)
ST08_408_Y54_0.sInit.InstName            :='ST08_408_Y54_0';
ST08_408_Y54_0.sInit.BitName            :='+8-408_Y54.0';
ST08_408_Y54_0.sInit.Description         :='Rückhaltezylinder li.+re. Auslauf STN8 AST';
ST08_408_Y54_0.sInit.HomePosDefine       :=HOME_INIT;(*HOME_ALWAYS;*)
ST08_408_Y54_0.sInit.InitDescription     :='GS einfahren';
ST08_408_Y54_0.sInit.WorkDescription     :='AS ausfahren';
ST08_408_Y54_0.sInit.DampBothTime        :=200;
ST08_408_Y54_0.sInit.KindOfValve         :='2G';
ST08_408_Y54_0.sInit.MaxTime             :=3000;

(* Init ST08_408_Y54_2 Abstapelzylinder 1 STN8 AST (Valve) *)
ST08_408_Y54_2.sInit.InstName            :='ST08_408_Y54_2';
ST08_408_Y54_2.sInit.BitName            :='+8-408_Y54.2';
ST08_408_Y54_2.sInit.Description         :='Aufstapelzylinder 1 STN8 AST';
ST08_408_Y54_2.sInit.HomePosDefine       :=HOME_INIT;
ST08_408_Y54_2.sInit.InitDescription     :='GS einfahren';
ST08_408_Y54_2.sInit.WorkDescription     :='AS ausfahren';
ST08_408_Y54_2.sInit.DampBothTime        :=200;
ST08_408_Y54_2.sInit.KindOfValve         :='2G';
ST08_408_Y54_2.sInit.MaxTime             :=3000;

(* Init ST08_408_Y54_4 Abstapelzylinder 2 STN8 AST (Valve) *)
ST08_408_Y54_4.sInit.InstName            :='ST08_408_Y54_4';
ST08_408_Y54_4.sInit.BitName            :='+8-408_Y54.4';
ST08_408_Y54_4.sInit.Description         :='Aufstapelzylinder 2 STN8 AST';
ST08_408_Y54_4.sInit.HomePosDefine       :=HOME_INIT;
ST08_408_Y54_4.sInit.InitDescription     :='GS einfahren';
ST08_408_Y54_4.sInit.WorkDescription     :='AS ausfahren';
ST08_408_Y54_4.sInit.DampBothTime        :=200;
ST08_408_Y54_4.sInit.KindOfValve         :='2G';
ST08_408_Y54_4.sInit.MaxTime             :=3000;

(* Rüstsatz Förderband Vereinzelner (Valve) *)
ST08_412_Y55_0.sInit.InstName            :='ST08_412_Y55_0';
ST08_412_Y55_0.sInit.BitName            :='+8-412_Y55.0';
ST08_412_Y55_0.sInit.Description         :='Rüstsatz Förderband Vereinzelner';
ST08_412_Y55_0.sInit.HomePosDefine       :=HOME_ALWAYS;
ST08_412_Y55_0.sInit.InitDescription     :='GS einfahren';
ST08_412_Y55_0.sInit.WorkDescription     :='AS ausfahren';
ST08_412_Y55_0.sInit.DampBothTime        :=200;
ST08_412_Y55_0.sInit.KindOfValve         :='2G';
ST08_412_Y55_0.sInit.MaxTime             :=3000;

(* Rüstsatz Förderband Stopper (Valve) *)
ST08_412_Y55_2.sInit.InstName            :='ST08_412_Y55_2';
ST08_412_Y55_2.sInit.BitName            :='+8-412_Y55.2';
ST08_412_Y55_2.sInit.Description         :='Rüstsatz Förderband Stopper';
ST08_412_Y55_2.sInit.HomePosDefine       :=HOME_ALWAYS;
ST08_412_Y55_2.sInit.InitDescription     :='GS einfahren';
ST08_412_Y55_2.sInit.WorkDescription     :='AS ausfahren';
ST08_412_Y55_2.sInit.DampBothTime        :=200;
ST08_412_Y55_2.sInit.KindOfValve         :='2G';
ST08_412_Y55_2.sInit.MaxTime             :=3000;
END_PROGRAM

(* POU Stations/ST_03_Ruestsaetze/ST_03_PRGs/ST03_Band_alt, ST *)
PROGRAM ST03_Band_alt
VAR_INPUT
	b_MoveRel 		:BOOL;
	fb_ton_Stopp_Band					: TON;
	bLockBand : BOOL;
END_VAR
VAR
	b_PosBetrieb	:BOOL;
	fb_rTrig_Off		: R_TRIG;
	fb_rTrig_stop		: R_TRIG;
	fb_ton_Off			: TON;
	fb_ton_Off2			: TON;
	fb_rTrig_On			: R_TRIG;
	fb_ton_Stau			: TON;
	fb_ton_Stau2		: TON;
	fb_rtrig_Stopp_Band	: R_TRIG;

	fb_rTrig_MoveRel	: R_TRIG;

	MsgOK				: BOOL;
	MsgCancel			: BOOL;
	lr_PT				: LREAL;
END_VAR
fb_ton_Stopp_Band(IN:= ,PT:=t#10m , Q=> , ET=> );																	(*Stop Wenn von der Sritzguss kein Teile kommen*)

fb_rtrig_Stopp_Band(CLK:=ST00_72_X1_3.BitInToCheck OR ST02_FDB_80_B02.BitInToCheck);
IF	fb_rtrig_Stopp_Band.Q THEN
	fb_ton_Stopp_Band.IN:=FALSE;
END_IF

(*Störung Oriental Motor bei SG-Maschine 3621*)
IF MP.ST03.SGM_3621 THEN
	IF NOT St03_V2.BitInToCheck THEN
		ST03_A5.SetSignalLow := TRUE;

		MessageHandler.Msg.ID:='PM101';
		MessageHandler.Msg.Color:=Color.red;
		MessageHandler.Msg.Name:='Error Förderband';
		MessageHandler.Msg.Text:='Störung Motor Oriental Förderband!';
		MessageHandler.Msg.Station:=3;

		MessageHandler(
			Prio:=2, 							(*1=highest, .. , 4=lowest*)
			Btn1Addr:=ADR(MsgOk),				(*Address of Button1 , if Zero then Button is unvisible*)
			Btn2Addr:=0(*ADR(MsgCancel)*),		(*Address of Button2 , if Zero then Button is unvisible*)
			sVisu:=Visu.Message);
	END_IF
END_IF
(*Motorregelung einschalten=========================================================== *)

IF NOT MP.ST03.SGM_3621 THEN
	IF  NOT ST03_51_M1.Error_ THEN
		IF	(NOT Safety_Fuses_AirPressure.SafetyOK OR gRunEmpty) AND
			ST03_51_M1.on THEN
			ST03_51_M1.MotorOff :=TRUE;
		END_IF

		IF	ModeSelect.Mode > MODE_MANUAL AND
			NOT gRunEmpty AND
			Safety_Fuses_AirPressure.SafetyOK AND
			NOT ST03_51_M1.on THEN
			ST03_51_M1.MotorOn :=TRUE;
		END_IF
	END_IF
END_IF

(*Fahren bis zu Flügelkamera Förderband============================================================ *)

IF	gTypeCode=312  OR		(*93pol*)
	gTypeCode=4991 THEN	(*102pol*)
	b_PosBetrieb:=TRUE;
	(*Impolsbetrieb Förderband============================================================ *)

	IF 	ST03_IFM_Camera.State=STATE_WAIT OR
 		ModeSelect.Mode>=MODE_MANUAL OR
		NOT MP.ST00.IFMCameraActive THEN

		fb_rTrig_MoveRel(CLK:= ST03_51_M1.Ready AND
								b_MoveRel);

		IF	fb_rTrig_MoveRel.Q THEN
			ST03_51_M1.sVelo.maxRpm;
			ST03_51_M1.Vorgabe_Velo:=16000; 			(*mm/min*)
			ST03_51_M1.Vorgabe_Pos_Rel:=MP.ST02.IFMPos;
			ST03_51_M1.MoveRel:=TRUE;
		END_IF

	END_IF

ELSE
	(*Dauerbetrieb Förderband============================================================ *)
	b_PosBetrieb:=FALSE;
	fb_ton_Off(IN:=ST00_73_K3.BitOutToSet , PT:=t#5m, Q=> , ET=> );			(*Stop Wenn von der SG-Maschine keine Teile kommen*)

	IF  gTypeCode = 322 THEN (*160pol*)
		fb_ton_Off2(IN:=ST00_73_K3.BitOutToSet AND								(* Schnittstelle Förderband frei für Spritzmaschine*)
						ST03_422_B64_4.BitInToCheck AND						(* Teil auf Abholposition Roboter *)
						(Robot01.ActualArea<>4), PT:=t#5s , Q=> , ET=> ); 			(*anhalten wenn Roboter nicht in der WT Area ist, die Ablageposition leer und die Abholposition voll ist*)
	ELSE
		fb_ton_Off2(IN:=ST00_73_K3.BitOutToSet AND								(* Schnittstelle Förderband frei für Spritzmaschine*)
						ST08_412_B59_0.BitInToCheck AND						(* Teil auf Abholposition Roboter *)
						(Robot01.ActualArea<>4), PT:=t#3s , Q=> , ET=> ); 		(*anhalten wenn Roboter nicht in der WT Area ist, die Ablageposition leer und die Abholposition voll ist*)
	END_IF

	IF gTypeCode = 5841 THEN	(*268pol*)
		(*Stop wenn 4 Teile auf unterer Führungsschiene belegt sind *)
		fb_ton_Stau2(IN:=	ModeSelect.Mode > MODE_MANUAL AND
							ST03_556_B69_5.BitInToCheck AND	(* Führungsschiene Überwachung Staustrecke*)
							(ST03_556_B69_7. BitInToCheck OR	(* ISK anwesend an Abholposition*)
							Robot01.ActualArea <> 0	AND		(* Roboter zw. Abhol- und Park-Pos.*)
							Robot01.ActualArea <> 5 	AND		(* Blister Pos*)
							Robot01.ActualArea <> 6	), 			(* Park-Pos.*)
							PT:=t#500ms , Q=> , ET=> );
	ELSE
		IF  MP.ST03.SGM_3621 THEN
			fb_ton_Stau.PT:=t#15s;
		ELSE
			lr_PT:=(112-MP.ST02.Override_Band) *0.25;
			fb_ton_Stau.PT:=LREAL_TO_TIME(lr_PT * 1000);
		END_IF
	
		fb_ton_Stau(IN:=	NOT ST00_73_K3.BitOutToSet AND
							Robot01.ActualArea <> 4 AND
							(ModeSelect.Mode = MODE_AUTO_RUN OR ModeSelect.Mode = MODE_AUTO_STOP) ,
							Q=> , ET=>); 			(*Stop wenn Teile nach dem Ablegen nicht weiter gefördert werden*)
	END_IF

	fb_rTrig_Off(CLK:= ModeSelect.Mode<=MODE_MANUAL );

	fb_rTrig_stop(CLK:= ModeSelect.Mode<=MODE_MANUAL AND ST03_51_M1.sVisuAxis.BtnStop.Pressed );

	fb_rTrig_On(CLK:= 	ModeSelect.Mode>MODE_MANUAL AND
						Safety_Fuses_AirPressure.SafetyOK );

	IF NOT MP.ST03.SGM_3621 THEN
		IF	fb_rTrig_On.Q THEN
			ST03_51_M1.MotorOn:=TRUE;
		END_IF

		IF	ST03_51_M1.On THEN
			ST03_51_M1.MoveP:=MP.ST03.BandMoveP;
			ST03_51_M1.MoveN:=NOT MP.ST03.BandMoveP;
		END_IF

		IF 	NOT DummyTest_160pol AND
			(fb_rTrig_Off.Q OR
			fb_ton_Off2.Q OR
			fb_ton_Off.Q OR
			fb_ton_Stau.Q OR
			fb_ton_Stau2.Q OR
			fb_rTrig_stop.Q OR
			bLockBand) THEN
			ST03_51_M1.MotorOn:=FALSE;
			ST03_51_M1.MotorOff:=TRUE;
			ST03_51_M1.MoveN:=FALSE;
			ST03_51_M1.MoveP:=FALSE;
		ELSIF
			DummyTest_160pol AND NOT SpecialMode06.startBand THEN
			ST03_51_M1.MotorOn:=FALSE;
			ST03_51_M1.MotorOff:=TRUE;
			ST03_51_M1.MoveN:=FALSE;
			ST03_51_M1.MoveP:=FALSE;
		END_IF
	ELSE

		(*Ansteuerung Oriental Motor bei SG-Maschine 3621*)

		IF	NOT Safety_Fuses_AirPressure.SafetyOK THEN
			ST03_A5.SetSignalLow:=TRUE;
			ST03_A5.SetSignalHigh :=FALSE;
		ELSIF
			fb_rTrig_Off.Q OR fb_ton_Off2.Q OR fb_ton_Stau.Q THEN
			ST03_A5.SetSignalLow := TRUE;
			ST03_A5.SetSignalHigh :=FALSE;
		ELSIF
			ModeSelect.Mode >MODE_MANUAL AND
			Safety_Fuses_AirPressure.SafetyOK THEN
			ST03_A5.SetSignalHigh :=TRUE;
			ST03_A5.SetSignalLow := FALSE;
		END_IF
	END_IF


END_IF
END_PROGRAM

(* POU zLibrary/ept/Sprache/ST_SwitchLng, ST *)
PROGRAM ST_SwitchLng
VAR_OUTPUT
	b_EndChangeLng		: BOOL;
END_VAR
VAR
	fb_state_entry			: ST_StateEntry;
	s_sprache			: STRING(10);
	b_first_cycle			: BOOL := TRUE;

	btn_Language		: ARRAY [0..3] OF sButtonVisu;

	fbTon_ChangeLng		: TON;
END_VAR
VAR_TEMP
	i					:INT;
END_VAR
fbTon_ChangeLng(
	IN:=	ST_ReadXmlLineMsg.b_EndChangeLng AND
		ST_ReadXmlLine.b_EndChangeLng,
	PT:= t#200ms,
	Q=> b_EndChangeLng,
	ET=> );

IF 	b_first_cycle THEN
	IF	fb_state_entry.fb_ton_Step.ET > t#15s OR
		MP.ST00.Sprache <>'' THEN
		s_sprache := MP.ST00.Sprache;
		CURRENTLANGUAGE:=MP.ST00.Sprache;
		b_first_cycle := FALSE;
	END_IF
ELSE
	MP.ST00.Sprache := CURRENTLANGUAGE;
END_IF
Btn_Init();

IF		btn_Language[1].Pressed THEN
		CURRENTLANGUAGE:= 'DE';
ELSIF
		btn_Language[2].Pressed THEN
		CURRENTLANGUAGE:= 'EN';
ELSIF
		btn_Language[3].Pressed THEN
		CURRENTLANGUAGE:= 'CZ';
END_IF


(* ======================================Schrittkette======================================== *)
fb_state_entry(i16_pos:= 1);

CASE fb_state_entry.i16_step OF
(*=======================================================*)
	INIT_OBJ:

		fb_state_entry.i16_next_step := 10;

(*=======================================================*)
	INIT:
			;

END_CASE

fb_state_entry(i16_pos:= 2 );
END_PROGRAM
ACTION Btn_Init:
btn_Language[1].Text:='DE';
btn_Language[2].Text:='EN';
btn_Language[3].Text:='CZ';

FOR i := 0 TO 3  BY 1DO
	btn_Language[i].Enable:=TRUE;
	btn_Language[i].BackgroundColor:=Color.lightgrey;
	btn_Language[i].TextColor:=Color.black;
	btn_Language[i].Visible:= TRUE;

END_FOR


IF	CURRENTLANGUAGE = 'DE' THEN
	i:=1;
ELSIF
	CURRENTLANGUAGE = 'EN' THEN
	i:=2;
ELSIF
	CURRENTLANGUAGE = 'CZ' THEN
	i:=3;
ELSE
	i:=1;
END_IF

btn_Language[i].BackgroundColor:=Color.grey;
END_ACTION

(* POU Stations/ST_02_RT_Tampondrucker/ST02_FBs/FB_Schwenken, ST *)
FUNCTION_BLOCK FB_Schwenken
VAR_INPUT
	b_quitt						: BOOL;
	b_0_grad					: BOOL;
	b_180_grad					: BOOL;
	b_90_grad					: BOOL;

END_VAR
VAR_IN_OUT
	ST02_90_180					: FB_Valve; 			(* 90 - 180 Grad (Valve) *)
	ST02_90_0					: FB_Valve; 			(* 90 - 0 Grad (Valve) *)
	ST02_90						:FB_ValveSensor;		 (* Schwenkarm 1 90 Grad*)
END_VAR

VAR_OUTPUT

	b_ready						: BOOL;
	b_done						: BOOL;
	b_busy						: BOOL;
	b_error						: BOOL;

	ST02_90_0_sens				: BOOL; 		(* 90 - 0 Grad (Sensor) *)
	ST02_90_sens				: BOOL;		(* 90 Grad (Sensor)*)
	ST02_90_180_sens			: BOOL; 		(* 90 - 180 Grad (Sensor) *)

END_VAR
VAR
	b_first_cycle						: BOOL := TRUE;
	fb_ton_wz						: TON;
	fb_ton_uez						: TON;
	fb_ton_quitt						: TON;
	fb_state_entry						: ST_StateEntry;
	fb_r_trig_start						: R_TRIG;
	fb_r_trig_init						: R_TRIG;
END_VAR

VAR_OUTPUT

END_VAR
VAR

END_VAR
IF b_first_cycle THEN
	b_first_cycle := FALSE;
END_IF

(* Zeiten *)
fb_ton_wz(IN:= , PT:= , Q=>  , ET=> );
fb_ton_uez(IN:= , PT:=DINT_TO_TIME(ST02_90_180.sInit.MaxTime * 4)  , Q=>  , ET=> );
fb_ton_quitt(IN:= , PT:= t#100ms, Q=> , ET=> );

ST02_90_0_sens:=ST02_90_0.SensorWorkIn[1].SensorSignal ; 				(* 90 - 0 Grad (Sensor) *)
ST02_90_sens:=ST02_90.ValveSensor;									(* 90 Grad (Sensor) *)
ST02_90_180_sens:=ST02_90_180.SensorWorkIn[1].SensorSignal; ; 			(* 90 - 180 Grad (Sensor) *)

(* Flanken *)
fb_r_trig_start(CLK:= b_0_grad OR b_90_grad OR b_180_grad, Q=> );

b_error := ST02_90_0.State < 0 OR ST02_90_180.State < 0;

IF	b_error THEN
	fb_state_entry.i16_next_step := FEHLER;
END_IF

fb_r_trig_init(CLK:=ModeSelect.Mode<=MODE_MANUAL);
IF	fb_r_trig_init.Q THEN
	fb_state_entry.i16_next_step := INIT;
END_IF

(* ==================================Schrittkette================================ *)
fb_state_entry(i16_pos:= 1, );

CASE fb_state_entry.i16_step OF
(*=======================================================*)
	INIT_OBJ:
		fb_state_entry.i16_next_step := INIT;


(*=======================================================*)
	INIT:
		IF fb_state_entry.E THEN
			fb_ton_wz.IN := FALSE;
			fb_ton_uez.IN := FALSE;
			b_ready := FALSE;
			b_done := FALSE;
			b_busy := FALSE;
			b_0_grad := FALSE;
			b_90_grad := FALSE;
			b_180_grad := FALSE;
		END_IF

		(*-----------------------Weiterschaltbedingungen----------------------------*)
		fb_state_entry.i16_next_step := BEREIT;

(*=======================================================*)
	BEREIT:
		IF fb_state_entry.E THEN
			b_ready := TRUE;
		END_IF

		(*-----------------------Weiterschaltbedingungen----------------------------*)
			IF 	fb_r_trig_start.Q  AND NOT b_error THEN
				IF	b_0_grad THEN
					fb_state_entry.i16_next_step := 110;
				ELSIF b_90_grad THEN
					fb_state_entry.i16_next_step := 200;
				ELSIF b_180_grad THEN
					fb_state_entry.i16_next_step := 300;
				END_IF
			END_IF

		IF fb_state_entry.X THEN
			b_busy := TRUE;
			b_done := FALSE;
			b_0_grad := FALSE;
			b_90_grad := FALSE;
			b_180_grad := FALSE;
			fb_ton_uez.IN:=FALSE;
		END_IF

(*=======================================================*)
	110:(*auf 0 Grad*)

		ST02_90_180.MoveInit:=TRUE;		(*Schwenkarm 1 drehen 90 - 180 Grad (Valve) *)
		ST02_90_0.MoveWork:=TRUE;	 	(*Schwenkarm 1 drehen 90 - 0 Grad (Valve) *)
		fb_state_entry.i16_next_step := 120;

	120:
		IF 	fb_state_entry.E THEN
			fb_ton_uez.IN:=TRUE;
		END_IF

		(*-----------------------Weiterschaltbedingungen----------------------------*)
		IF 	(ST02_90_180.State =STATE_OK AND
			ST02_90_0.State =STATE_OK) OR
			ST02_90_0.SensorWorkIn[1].SensorSignal   THEN
			b_done := TRUE;
			b_busy := FALSE;
			fb_state_entry.i16_next_step := BEREIT;
		END_IF

		IF	fb_ton_uez.Q THEN
			fb_state_entry.i16_next_step := FEHLER;
		END_IF

		IF fb_state_entry.X THEN
			fb_ton_uez.IN:=FALSE;
		END_IF

(*=======================================================*)
	200:(*auf 90 Grad*)

		ST02_90_180.MoveInit:=TRUE;		(*Schwenkarm 1 drehen 90 - 180 Grad (Valve) *)
		ST02_90_0.MoveInit:=TRUE;	 		(*Schwenkarm 1 drehen 90 - 0 Grad (Valve) *)
		fb_state_entry.i16_next_step := 210;

	210:
		IF 	fb_state_entry.E THEN
			fb_ton_uez.IN:=TRUE;
		END_IF

		(*-----------------------Weiterschaltbedingungen----------------------------*)
		IF 	(ST02_90_180.State =STATE_OK AND
			ST02_90_0.State =STATE_OK) OR
			ST02_90.ValveSensor THEN
			b_done := TRUE;
			b_busy := FALSE;
			fb_state_entry.i16_next_step := BEREIT;
		END_IF

		IF	fb_ton_uez.Q THEN
			fb_state_entry.i16_next_step := FEHLER;
		END_IF

		IF fb_state_entry.X THEN
			fb_ton_uez.IN:=FALSE;
		END_IF

(*=======================================================*)
	300:(*auf 0 Grad*)

		ST02_90_180.MoveWork:=TRUE;		(*Schwenkarm 1 drehen 90 - 180 Grad (Valve) *)
		ST02_90_0.MoveInit:=TRUE;	 		(*Schwenkarm 1 drehen 90 - 0 Grad (Valve) *)
		fb_state_entry.i16_next_step := 310;

	310:
		IF 	fb_state_entry.E THEN
			fb_ton_uez.IN:=TRUE;
		END_IF

		(*-----------------------Weiterschaltbedingungen----------------------------*)
		IF 	(ST02_90_180.State =STATE_OK AND
			ST02_90_0.State =STATE_OK) OR
			ST02_90_180.SensorWorkIn[1].SensorSignal   THEN
			b_done := TRUE;
			b_busy := FALSE;
			fb_state_entry.i16_next_step := BEREIT;
		END_IF

		IF	fb_ton_uez.Q THEN
			fb_state_entry.i16_next_step := FEHLER;
		END_IF

		IF fb_state_entry.X THEN
			fb_ton_uez.IN:=FALSE;
		END_IF
(*=======================================================*)
	FEHLER:
		IF fb_state_entry.E THEN
			b_error := TRUE;
			fb_ton_quitt.IN := FALSE;
		END_IF

		(*-----------------------Weiterschaltbedingungen----------------------------*)
		IF  NOT fb_state_entry.E AND NOT b_error THEN
			fb_ton_quitt.IN := TRUE;
		END_IF

		IF fb_ton_quitt.Q THEN
			fb_ton_quitt.IN := FALSE;
			fb_state_entry.i16_next_step := INIT;
		END_IF

(*=======================================================*)
	STOP:
		IF fb_state_entry.E THEN
			fb_ton_quitt.IN := FALSE;
		END_IF

		(*-----------------------Weiterschaltbedingungen----------------------------*)
		IF b_quitt AND NOT fb_state_entry.E THEN
			fb_ton_quitt.IN := TRUE;
		END_IF

		IF fb_ton_quitt.Q THEN
			fb_ton_quitt.IN := FALSE;
			fb_state_entry.i16_next_step := INIT;
		END_IF

END_CASE

fb_state_entry(i16_pos:= 2 );
END_FUNCTION_BLOCK

(* POU zLibrary/Valve/FB_Valve, ST *)
FUNCTION_BLOCK FB_Valve (*01.DEZ 2010,  B.Happach*)
VAR_OUTPUT
	State					: StateObject;		(* State of the object *)
	HomePosition			: BOOL;				(* object in home-position*)
	InitPosition				: BOOL;				(* Reflectet SensorState - All sensors showing "Init" *)
	WorkPosition			: BOOL;				(* Reflectet SensorState - All sensors showing "Work" *)
	ValveWorkOut			: ARRAY[1..8] OF sValveSensor_ValveOut; (* Structure To Sensorobject - Index is set in Init from Sensor *)
	ValveInitOut				: ARRAY[1..8] OF sValveSensor_ValveOut; (* Structure To Sensorobject - Index is set in Init from Sensor *)

END_VAR
VAR_INPUT
	MoveWork				: BOOL; 			(* Move to Workposition *)
	MoveInit				: BOOL;				(* Move to Initposition *)
	Enable					: BOOL:=TRUE;		(* Enables the operations on the valve *)
	Reset					: BOOL; 			(* switch for resetting the object *)
	SFCCurrentStep			: STRING(80);		(* aktually step in the step flow chart *)
	SFCCurrentPOU			: STRING(80);		(* Name of the step flow chart *)
	sInit						: sValveInit;			(* Initializingvalues to the Instance *)
	strAnlayse				: STRING(255); 		(*String to analyse Lockings*)
	SensorWorkIn			: ARRAY[1..8] OF sValveSensor_SensorOut; (* States from Worksensors - Index is set in Init from Sensor *)
	SensorInitIn				: ARRAY[1..8] OF sValveSensor_SensorOut; (* States from Initsensors - Index is set in Init from Sensor *)
	fb_Ton_Reset			:TON;
	fb_rTrig_Reset			:R_TRIG;
	WorkPos				:BOOL;
	InitPos					:BOOL;
	i						:INT;
END_VAR
VAR_IN_OUT
	sVisu					: sValveVisu;   		(* Structure for Visualisation *)
END_VAR
VAR
	CoilA					AT %Q* : BOOL; 	(* For Moving to WorkPosition *)
	CoilB					AT %Q* : BOOL; 	(* For Moving to InitPosition *)
	CoilAState				: BOOL; 			(* State Of Coil A - Depending on Valvetype *)
	CoilBState				: BOOL; 			(* State Of Coil B - Depending on Valvetype *)

(* Init and Worksensor Handling *)
	NoOfWorkSensors			: DINT;			(* Counter of Worksensors - Incremented by Sensorobject while initialisation *)
	NoOfInitSensors				: DINT;			(* Counter of Initsensors - Incremented by Sensorobject while initialisation *)
	NoOfValveCoils				: DINT;			(* Number of ValveCoils - from Init Struct *)

	IdxWork					: DINT;			(* Index Variable use in For-Loops *)
	IdxInit						: DINT;			(* Index Variable use in For-Loops *)

	HiCountWork				: DINT;			(* Varibable To Cout Sensors wich are high *)
	LoCountWork				: DINT;			(* Varibable To Cout Sensors wich are low *)
	HiCountInit					: DINT;			(* Varibable To Cout Sensors wich are high *)
	LoCountInit					: DINT;			(* Varibable To Cout Sensors wich are low *)

	WorkSensors_AllHi			: BOOL;			(* Internal Used Flag  *)
	WorkSensors_AllLo			: BOOL;			(* Internal Used Flag  *)
	InitSensors_AllHi				: BOOL;			(* Internal Used Flag  *)
	InitSensors_AllLo			: BOOL;			(* Internal Used Flag  *)
(* Movement Handling *)
	WorkingStep				: DINT;			(* Index for StateMachine *)
	MoveWorkStored			: BOOL; 		(* Stored Command "Move to Workposition"  *)
	MoveInitStored				: BOOL;			(* Stored Command "Move to Initposition" *)

	DampBoth					: BOOL;			(* This flag is Set when Damp both is required and possible *)
	DampBothTimer				: TON;			(* This Timer is used to set both valvecoils to fill the zylinder from Both sides *)

	DfltTxtDescription			: STRING(80):='Not defined!';
	DfltTxtVisuWorkButtonText 	: STRING(80):='Work';
	DfltTxtVisuInitButtonText 	: STRING(80):='Init';

(* Init Handling *)
	InitStep						: INT;				(* Init Step StateMachine *)
	InstanceNo					: INT;				(* Instance No for Language Handling - Used for Global Class functions *)
	InitState						: BOOL :=	FALSE;	(* Internal State for initialising *)

(* Visu Handling *)
	BtnMoveWork				: VisuButton;		(* Manage button *)
	BtnMoveInit					: VisuButton;		(* Manage button *)
	BtnReset					: VisuButton;		(* Manage button *)


(* Error Handling *)
	TimerTimeOut				: CheckProcTime;	(* Timer generates timeout signal *)
	ProcessTime				: DINT;				(* Counts the time since starting operation *)

	Error						: ErrorStruct;
	ErrorElapsed				: R_TRIG;

	LaufschriftErrh				: FB_Laufschrift;
	LaufschriftObj				: FB_Laufschrift_STR255;
	LaufschriftAnalyse			: FB_Laufschrift_STR255;
	TempString					: STRING(255);

	FB_ReadXmlLineConf		: FB_ReadXmlLine;
	FB_ReadXmlLineMsg		 : FB_ReadXmlLine;

END_VAR


(*Description kind of valve:
-------------------------------------
A	:	Valve with 1 coil  3/2 or 5/2 monostable
B	:	Valve with 2 coils 5/2 impulse
2G	:	Valve with 2 coils 2x 3/2
======================================*)

							
Error.No:=0;
Error.Text:='';

(*ermittel wo der Zylinder steht und schaltet das Ventil nach dem Reset auf die Position wo der Zylinder steht*)
WorkPos:=TRUE;
FOR i:=1 TO DINT_TO_INT(NoOfWorkSensors)  BY 1 DO
	IF	NOT SensorWorkIn[i].SensorSignal AND WorkPos THEN
		WorkPos:=FALSE;
	END_IF
END_FOR

InitPos:=TRUE;
FOR i:=1 TO DINT_TO_INT(NoOfInitSensors)  BY 1 DO
	IF	NOT SensorInitIn[i].SensorSignal AND InitPos THEN
		InitPos:=FALSE;
	END_IF
END_FOR
fb_Ton_Reset(IN:=NOT Reset, PT:=t#200ms);
fb_rTrig_Reset(CLK:=fb_Ton_Reset.Q);
IF	fb_rTrig_Reset.Q THEN
	MoveWork	:=WorkPos AND NoOfWorkSensors > 0; 			(* Move to Workposition *)
	MoveInit	:=InitPos AND NoOfInitSensors > 0; 				(* Move to Initposition *)
END_IF

(*------------------------------------------------------------------
	Initialization
  ------------------------------------------------------------------*)
IF 	NOT InitState THEN
	CASE InitStep OF

	0: (* Init Instance *)
			InitStep:=1;
	1: (* Init Internal OjbNo *)
			gValve.ObjCount:=gValve.ObjCount+1;
			InstanceNo:=gValve.ObjCount;
			InitStep:=50;

	50: (*Check KindOfValve*)
		IF 	sInit.KindOfValve='A' THEN
			NoOfValveCoils:=1;
			InitStep:=100;
		ELSIF
			sInit.KindOfValve='B' OR
			sInit.KindOfValve='2G' THEN
			NoOfValveCoils:=2;
			InitStep:=100;
		ELSE
			InitState:=FALSE;
			State:=STATE_ERROR;
			FB_ReadXmlLineMsg.ID:='KindOfValve';
			Error.No:=3;
			Error.Text:=sInit.InstName;
			Error.Text:=CONCAT(Error.Text,': ');
			Error.Text:=CONCAT(Error.Text,sInit.Description);
			Error.Text:=CONCAT(Error.Text,' - ');
			Error.Text:=CONCAT(Error.Text,FB_ReadXmlLineMsg.Text);
		END_IF

	100: (* Init Done *)
		InitState:=TRUE;
	END_CASE

END_IF (*InitState = FALSE*)

(* Add InitState to Global-Init-State to collect all Objects *)
gInitCollect:=gInitCollect AND InitState;

IF 	gInitOk THEN

	sVisu.Description			:= DfltTxtDescription;
	sVisu.WorkDescription		:= DfltTxtVisuWorkButtonText;
	sVisu.InitDescription			:= DfltTxtVisuInitButtonText;
(*------------------------------------------------------------------
	Show and Read Visu Buttons
  ------------------------------------------------------------------*)
	BtnMoveWork(Button:=sVisu.BtnMoveWork,
							Enable:= ModeSelect.Mode=MODE_MANUAL AND
									Enable AND
									(sInit.KindOfValve<>'2G' AND
									 NOT WorkPosition OR sInit.KindOfValve='2G' AND
									(NOT WorkPosition OR NOT CoilA)		) AND
									(State=STATE_WAIT OR State=STATE_ERROR),
							TextOn:=sVisu.WorkDescription
							);

	BtnMoveInit(Button:=sVisu.BtnMoveInit,
							Enable:=		ModeSelect.Mode=MODE_MANUAL AND
											Enable AND
											(	sInit.KindOfValve<>'2G' AND
												NOT InitPosition OR
												sInit.KindOfValve='2G' AND
											( 	NOT InitPosition OR NOT CoilB)		) AND
											(State=STATE_WAIT OR State=STATE_ERROR),
							TextOn:=sVisu.InitDescription
							);

	BtnReset(		Button:=sVisu.BtnReset,
							Enable:=ModeSelect.Mode=MODE_MANUAL ,
							TextOn:='Reset',
							);
END_IF

(*------------------------------------------------------------------
	Manual Mode
  ------------------------------------------------------------------*)
IF ModeSelect.Mode=MODE_MANUAL AND Enable THEN

	MoveWork:=MoveWork OR BtnMoveWork.Pressed;
	MoveInit:=MoveInit OR BtnMoveInit.Pressed;
	Reset:=Reset OR BtnReset.Pressed;
END_IF

(*------------------------------------------------------------------
	Sensor and Coil State Handling
  ------------------------------------------------------------------*)

(* Get States of All declarated Init Sensors *)
HiCountInit:=0;
LoCountInit:=0;
IF 	NoOfInitSensors>0 THEN
	FOR IdxInit:=1 TO NoOfInitSensors DO
		IF SensorInitIn[IdxInit].SensorSignal THEN
			HiCountInit:=HiCountInit+1;
		ELSE
			LoCountInit:=LoCountInit+1;
		END_IF
	END_FOR
END_IF
(* Get States of All declarated Work Sensors *)
HiCountWork:=0;
LoCountWork:=0;
IF 	NoOfWorkSensors>0 THEN
	FOR IdxWork:=1 TO NoOfWorkSensors DO
		IF SensorWorkIn[IdxWork].SensorSignal THEN
			HiCountWork:=HiCountWork+1;
		ELSE
			LoCountWork:=LoCountWork+1;
		END_IF
	END_FOR
END_IF

(* Handle Sensor States *)
InitSensors_AllHi:= (HiCountInit=NoOfInitSensors);
InitSensors_AllLo:= (LoCountInit=NoOfInitSensors);

WorkSensors_AllHi:= (HiCountWork=NoOfWorkSensors);
WorkSensors_AllLo:= (LoCountWork=NoOfWorkSensors);


(* Write Coilstates To Local Var - depending on Valvetype*)
IF 	NoOfValveCoils=1	THEN
	CoilAState:= CoilA;
	CoilBState:= NOT CoilA;
ELSE
		IF	sInit.KindOfValve='B' THEN
			IF 	NoOfWorkSensors>0 THEN
				CoilAState:=WorkSensors_AllHi AND InitSensors_AllLo ;
			ELSE
				CoilAState:=MoveWorkStored;
			END_IF

			IF 	NoOfInitSensors>0 THEN
				CoilBState:=InitSensors_AllHi AND WorkSensors_AllLo;
			ELSE
				CoilBState:=MoveInitStored;
			END_IF
		ELSE
			CoilAState:=CoilA AND NOT CoilB;
			CoilBState:=CoilB AND NOT CoilA;
		END_IF
END_IF

(* Handle Case if No Sensor Is declared *)
IF NoOfInitSensors>0 AND NoOfWorkSensors>0 THEN
	(* Work- and Initsensor available *)
	InitPosition:=InitSensors_AllHi AND WorkSensors_AllLo;
	WorkPosition:=WorkSensors_AllHi AND InitSensors_AllLo;
ELSIF
	NoOfInitSensors=0 AND NoOfWorkSensors>0 THEN
	(* Worksensor available and Initsensor NOT available *)
	WorkPosition:=WorkSensors_AllHi;
	InitPosition:=WorkSensors_AllLo AND CoilBState;
ELSIF
	NoOfInitSensors>0 AND NoOfWorkSensors=0 THEN
	(* Worksensor NOT available and Initsensor available *)
	InitPosition:=InitSensors_AllHi;
	WorkPosition:=InitSensors_AllLo AND CoilAState;
ELSIF
	NoOfInitSensors=0 AND NoOfWorkSensors=0 THEN
	(* If NO sensor is available then Inicate State over valvecoils*)
	InitPosition:=CoilBState;
	WorkPosition:=CoilAState;
END_IF

(*------------------------------------------------------------------
	Generate Damp Both Flag
  ------------------------------------------------------------------*)
DampBoth:=	sInit.KindOfValve='2G' AND
			sInit.DampBothTime>0 AND
			NOT (CoilA OR CoilB) AND
         			(   	MoveInit AND NOT InitPosition OR
             			MoveWork AND NOT WorkPosition );

(*------------------------------------------------------------------
	Move-Handling
  ------------------------------------------------------------------*)

CASE WorkingStep OF
	0: (* State STATE_WAIT *)

		IF	InitState THEN
			State:=STATE_WAIT;
			IF 	MoveWork OR
				MoveInit THEN
				WorkingStep:=100;
				TimerTimeOut.Start:=TRUE;
				State:=STATE_RUN;
				MoveWorkStored:=MoveWork;
				MoveInitStored:=MoveInit;
			END_IF
		END_IF

100:(* Move *)
		(* Check Damp Both *)
		IF DampBoth THEN
			WorkingStep:=110;
		ELSE
			WorkingStep:=120;
		END_IF
110:(* DampBoth *)
		DampBothTimer.IN:=TRUE;
		CoilA:=TRUE;
		CoilB:=TRUE;
		IF DampBothTimer.Q THEN
			WorkingStep:=120;
		END_IF
120: (* SET Valve Coils Move to Selected direction *)
		IF 	NoOfValveCoils=1 THEN
			CoilA:=MoveWorkStored;
			CoilB:=FALSE;
		ELSE
			CoilA:=MoveWorkStored;
			CoilB:=MoveInitStored;
		END_IF
		WorkingStep:=130;

